Beispiel Initialisierung:

(*Init ST08_180_M1 Abstapeln*)
ST08_180_M1.sConfig.Description		:='Abstapeln';
ST08_180_M1.sConfig.InstName			:='ST08_180_M1';
ST08_180_M1.sConfig.Aktiv				:=TRUE;
ST08_180_M1.sConfig.Skalierfaktor		:=0.00034332275390625	;	(*360 / 1048576*)
ST08_180_M1.sConfig.Getriebefaktor		:=10;
ST08_180_M1.sConfig.Modulo			:=FALSE;
ST08_180_M1.sConfig.Pos_Faktor		:=5;				(*Weg bei einer Umdrehung in mm (nach Getriebe)*)
ST08_180_M1.sConfig.maxRpm			:=5338;
ST08_180_M1.sConfig.ModeOfOperation	:=CSP;			(*CSP,CSV,CST,CSTCA muss an der KLemme (Coe-Online 7010.03) eingestellt werden*)
(*nur für Coe-Online 7010.03 (CSP) position mode*)
ST08_180_M1.sConfig.RampTime		:=t#500ms;		(*Bauselle*)(*Beschleunigung und Bremsrampe*)
ST08_180_M1.sConfig.PosDiffControl_on	:=FALSE;		(*Baustelle*)
ST08_180_M1.sConfig.max_PosDiff		:=720;			(*Baustelle*)
ST08_180_M1.sConfig.SW_Limit_on		:=FALSE;
ST08_180_M1.sConfig.SW_Limit_min		:=-1000;
ST08_180_M1.sConfig.SW_Limit_max	:=1000;
ST08_180_M1.sConfig.lr_kp 				:= 800;
ST08_180_M1.sConfig.lr_ki 				:= 100.0;
ST08_180_M1.sConfig.lr_kd 				:= 50;

Beispiel Aufruf::

(*Call ST08_180_M1 Abstapeln*)
ST08_180_M1			(	sVisu:=	Visu.ST08_180_M1,
						Override:=	 MP.ST08.Override_Abstapeln,
						Offset:=		MP.ST08.PosOffsetAbstapeln.Pos,	(* in mm oder Grad am Abtrieb*)
						Reset:=		Visu.ModeSelect.BtnReset.Pressed );
IF	ST08_180_M1.sVisuAxis.BtnTeach.Pressed THEN
	TD.PosAbstapeln[ST08_180_M1.sVisuAxis.PosNr].Pos:= ST08_180_M1.sctrl.in.Position;
END_IF


 ===============================================================================================================================*)
END_ACTION
ACTION sub_connect:
IF	e_Toggle <> sHelp.b_ToggleHelp OR	(*die alten EL7211 haben kein e_Toggle, desshalb gibt es auch den e_State*)
	e_State = 8 THEN
	Connect:=TRUE;
	sHelp.b_ToggleHelp:=e_Toggle;
ELSE
	Connect:=FALSE;
END_IF
e_State:=e_State;(*
0x___1 = Slave in 'INIT' state
0x___2 = Slave in 'PREOP' state
0x___3 = Slave in 'BOOT' state
0x___4 = Slave in 'SAFEOP' state
0x___8 = Slave in 'OP' state
0x001_ = Slave signals error
0x002_ = Invalid vendorId, productCode... read
0x004_ = Initialization error occurred
0x008_ = Slave disabled
0x010_ = Slave not present
0x020_ = Slave signals link error
0x040_ = Slave signals missing link
0x080_ = Slave signals unexpected link
0x100_ = Communication port A
0x200_ = Communication port B
0x400_ = Communication port C
0x800_ = Communication port D*)
END_ACTION
ACTION sub_ctrl:
(*================================================================================================*)
(*Statusword*)
(*Bit  0*) sCtrl.in.Ready_to_switch_on:=		e_Statusword.0;
(*Bit 1 *) sCtrl.in.Switched_on:=			e_Statusword.1;
(*Bit 2 *) sCtrl.in.Operation_enabled	:=	e_Statusword.2;
(*Bit 3 *) sCtrl.in.Fault:=					e_Statusword.3;
(*Bit 4 *) 								e_Statusword.4;
(*Bit 5 *) 								e_Statusword.5;
(*Bit 6 *) sCtrl.in.Switch_on_disabled:=		e_Statusword.6;
(*Bit 7 *) sCtrl.in.Warning:=				e_Statusword.7;
(*Bit 8 *) 								e_Statusword.8;
(*Bit 9 *) 								e_Statusword.9;
(*Bit 10*) sCtrl.in.TxPDOToggle:=			e_Statusword.10; (*An-/Abwahl über 0x8010:01[} 136]*)
(*Bit 11*) sCtrl.in.Internal_Limit_active:=		e_Statusword.11;
(*Bit 12*) sCtrl.in.Target_value_ignored:=	e_Statusword.12;
(*Bit 13*) 								e_Statusword.13;
(*Bit 14*) 								e_Statusword.14;
(*Bit 15*) 								e_Statusword.15;

(*Controlword*)
(*Bit 0 *) a_Controlword.0:= sCtrl.out.Switch_on;
(*Bit 1 *) a_Controlword.1:= sCtrl.out.Enable_voltage;
(*Bit 2 *) a_Controlword.2:= sCtrl.out.Shutdown;
(*Bit 3 *) a_Controlword.3:= sCtrl.out.Enable_operation;
(*Bit 4 *) a_Controlword.4;
(*Bit 5 *) a_Controlword.5;
(*Bit 6 *) a_Controlword.6;
(*Bit 7 *) a_Controlword.7:= sCtrl.out.Fault_reset;
(*Bit 8 *) a_Controlword.8;
(*Bit 9 *) a_Controlword.9;
(*Bit 10*) a_Controlword.10;
(*Bit 11*) a_Controlword.11;
(*Bit 12*) a_Controlword.12;
(*Bit 13*) a_Controlword.13;
(*Bit 14*) a_Controlword.14;
(*Bit 15*) a_Controlword.15;
END_ACTION
ACTION sub_fb:
(* Zeiten *)
sFb.ton_uez		(IN:= ,PT:= t#3000ms, Q=>, ET=> );

sFb.ton_uez_velo	(IN:= sVelo.dif >15 AND on, PT:= t#300ms, Q=> , ET=> );
sFb.r_trig_Auto(CLK:=ModeSelect.Mode>MODE_MANUAL);
sFb.r_trig_Hand(CLK:=ModeSelect.Mode=MODE_MANUAL);
IF	sFb.r_trig_Hand.Q THEN
	sVisuAxis.Control:=TRUE;
ELSIF
	sFb.r_trig_Auto.Q THEN
	sVisuAxis.Control:=FALSE;
END_IF

(* Flanken *)
sFb.r_trig_stop(CLK:= NOT sVisuAxis.BtnStop.Pressed );
sFb.r_trig_reset(CLK:=NOT sVisuAxis.BtnReset.Pressed );
sFb.r_trig_MotorOn(CLK:=NOT sVisuAxis.BtnMotorOn.Pressed);
sFb.r_trig_jogP(CLK:= NOT sVisuAxis.BtnJogP.Pressed);
sFb.r_trig_jogM(CLK:=NOT sVisuAxis.BtnJogM.Pressed);
sFb.r_trig_MoveP(CLK:= NOT MoveP);
sFb.r_trig_MoveM(CLK:=NOT MoveN);
sFb.r_trig_MoveAbs(CLK:= NOT sVisuAxis.BtnMoveAbs.Pressed);

(*
sFb.ton_quitt		(IN:= ,PT:= t#100ms, Q=> , ET=> );
sFb.r_trig_quitt(CLK:=
			NOT On AND (*FEHLER wird dadurch automatisch quittiert*)
			NOT Reset AND
			NOT sVisuAxis.BtnReset.Pressed );
*)


sFb.ton_quitt(
		IN:=	NOT On AND (*FEHLER wird dadurch automatisch quittiert*)
				NOT Reset AND
				NOT sVisuAxis.BtnReset.Pressed ,
		PT:= 	t#200ms);
sFb.r_trig_quitt(CLK:=sFb.ton_quitt.Q);
END_ACTION
ACTION sub_Pos:
sPos.ist:=sctrl.in.Position;
(*===============================================================================*)
IF	(*config.Modulo OR*)
	sConfig.Pos_Faktor=0 THEN
	sConfig.Pos_Faktor:=1;
END_IF

(*Encoderüberlauf===================================================================================*)
sPos.lr_delta_ueberlauf:=ABS(sPos.lr_akt_alt - e_Position);

IF	sPos.lr_akt_alt >	(sPos.r_32bit - sPos.lr_delta_ueberlauf) AND						(*Überlauf bei 4294967295*)
	e_Position < sPos.lr_delta_ueberlauf THEN
	sPos.i32_count_ueberlauf:=	sPos.i32_count_ueberlauf +1;
ELSIF sPos.lr_akt_alt < sPos.lr_delta_ueberlauf AND									(*Überlauf bei 4294967295*)
	e_Position >(sPos.r_32bit - sPos.lr_delta_ueberlauf) THEN
	sPos.i32_count_ueberlauf:=	sPos.i32_count_ueberlauf -1;
END_IF
sPos.lr_akt_alt:= e_Position;

sPos.lr_Uebrlauf_Dist:=sPos.r_32bit * sConfig.Skalierfaktor;							(*Pos in Grad am Motor*)
sPos.lr_Uebrlauf_Dist:=sPos.lr_Uebrlauf_Dist/ sConfig.Getriebefaktor;					(*Pos in Grad am Getriebe*)

IF	NOT sConfig.Modulo THEN
	sPos.lr_Uebrlauf_Dist:=sPos.lr_Uebrlauf_Dist * (sConfig.Pos_Faktor/360);			(* Position in mm bei Linearachse*)
END_IF
sPos.lr_Uebrlauf_DistOne:=sPos.lr_Uebrlauf_Dist;

(*Positon auf Null stellen wenn der Überlauf erreicht ist*)
IF	sPos.i32_count_ueberlauf < - sConfig.Getriebefaktor THEN
	sCtrl.out.Target_Position:=sCtrl.out.Target_Position + (sConfig.Getriebefaktor * sPos.lr_Uebrlauf_DistOne );
	sPos.i32_count_ueberlauf:=sPos.i32_count_ueberlauf + LREAL_TO_DINT(sConfig.Getriebefaktor);
ELSIF  sPos.i32_count_ueberlauf >  sConfig.Getriebefaktor THEN
	sCtrl.out.Target_Position:=sCtrl.out.Target_Position - (sConfig.Getriebefaktor * sPos.lr_Uebrlauf_DistOne );
	sPos.i32_count_ueberlauf:=sPos.i32_count_ueberlauf - LREAL_TO_DINT(sConfig.Getriebefaktor);
END_IF

sPos.lr_Uebrlauf_Dist:=sPos.lr_Uebrlauf_Dist *DINT_TO_LREAL(sPos.i32_count_ueberlauf);

(*Multiturn======================================================================================*)

sConfig.Skalierfaktor;
sCtrl.in.Position:=UDINT_TO_LREAL(e_Position )*sConfig.Skalierfaktor;	(*Pos in Grad am Motor*)
(*sPos.lr_Mod:=LMOD(sCtrl.in.Position ,config.Modulofaktor);		(*Moduloposition*)*)
sCtrl.in.Position:=sCtrl.in.Position/ sConfig.Getriebefaktor;					(*Pos in Grad am Getriebe*)
sPos.lr_Mod:=LMOD((sCtrl.in.Position-Offset) ,360);			(*Pos in Grad 0° - 360° *)

IF	NOT sConfig.Modulo THEN
	sCtrl.in.Position:=sCtrl.in.Position * (sConfig.Pos_Faktor/360);			(* Position in mm bei Linearachse*)

	sPos.lr_Target:=sCtrl.out.Target_Position / (sConfig.Pos_Faktor/360) ;	(*Pos in Grad am Getriebe° *)
	sPos.lr_Offset_Ink:=Offset / (sConfig.Pos_Faktor/360) ;		 (*OffsetPos in Grad am Getriebe° *)
ELSE
	sPos.lr_Target:=sCtrl.out.Target_Position;
END_IF

sCtrl.in.Position:=sPos.lr_Uebrlauf_Dist+sCtrl.in.Position-Offset;

sPos.lr_Target:=sPos.lr_Target * sConfig.Getriebefaktor;				(*Pos in Grad am Motor° *)
sPos.lr_Offset_Ink:=sPos.lr_Offset_Ink* sConfig.Getriebefaktor;			(*OffsetPos in Grad am Motor° *)
sPos.i32_Offset_Ink:=LREAL_TO_UDINT(sPos.lr_Offset_Ink / sConfig.Skalierfaktor);		(*OffsetPos in Inkrementen am Motor° *)
a_Target_Position:=LREAL_TO_UDINT(sPos.lr_Target / sConfig.Skalierfaktor);	(*Pos in Inkrementen am Motor° *)

a_Target_Position:=a_Target_Position-sPos.i32_Offset_Ink;
e_Position;


(*Singelturn===Baustelle========================================================================*)
sPos.lr_ModuloPosInc:=LMOD(e_Position ,sPos.r_20bit);			(*Moduloposition in Ikrementen*)

sPos.lr_ModuloHelp:=(e_Position - LREAL_TO_UDINT(sPos.lr_ModuloPosInc)) / LREAL_TO_UDINT(sPos.r_20bit) ;
sPos.lr_ModuloHelp2:=(e_Position - LREAL_TO_UDINT(sPos.lr_ModuloPosInc)) / LREAL_TO_UDINT(sPos.r_20bit) ;
sPos.i16_ModuloHelp:=GANZE_ZAHL(sPos.lr_ModuloHelp2 / sConfig.Getriebefaktor);
sPos.lr_ModuloCount:=sPos.lr_ModuloHelp2 - (sPos.i16_ModuloHelp * sConfig.Getriebefaktor);

sPos.lr_Pos:= (sPos.lr_ModuloCount * sPos.r_20bit)+sPos.lr_ModuloPosInc;
sPos.lr_Pos:=sPos.lr_Pos* sConfig.Skalierfaktor;				(*Pos in Grad am Motor*)
sPos.lr_Pos:=sPos.lr_Pos / sConfig.Getriebefaktor;				(*Pos in Grad am Getriebe*)
sPos.lr_Pos:=LMOD(sPos.lr_Pos ,360);							(*Pos in Grad 0° - 360° *)
sPos.lr_Pos:=sPos.lr_Pos * (sConfig.Pos_Faktor/360);			(* Position in mm bei Linearachse*)



(*Schleppfehler===================================================================================*)
sCtrl.in.Following_Error:=DINT_TO_LREAL(e_Following_Error)*sConfig.Skalierfaktor;

sFb.ton_aufPos(
		IN:= ABS(sCtrl.out.Target_Position - sCtrl.in.Position) <1,
		PT:=t#20ms,
		Q=>On_Position);
END_ACTION
ACTION sub_rec_Torque:
IF	ABS(e_Torque) > Torque[1] THEN
	i:=1;
	FOR i:=NO_OF_Torque TO 2 BY-1 DO
	   Torque[i] := Torque[i-1];
	END_FOR
	 Torque[1]:=ABS(e_Torque);
END_IF
END_ACTION
ACTION sub_Regler:
sPos.r_18bit;
sVelo.Faktor:=sPos.r_18bit / 60;
(*=============================================================================================================*)

sVelo.maxRpmNachGertiebe	:=sConfig.maxRpm/ sConfig.Getriebefaktor;		(*Maximale Drehzahl nach Getriebe*)
sVelo.maxLinear		:=sVelo.maxRpmNachGertiebe * sConfig.Pos_Faktor;		(*Maximale Geschwindigkeit in mm/min*)
IF	 sConfig.Modulo THEN
	sVelo.maxRpm:=sVelo.maxRpmNachGertiebe;	(*rpm*)
	sVelo.Vorgabe_Velo_rpm:=Vorgabe_Velo * LREAL_TO_INT(sConfig.Getriebefaktor);
ELSE
	sVelo.maxRpm:=sVelo.maxLinear;			(*mm/min*)
	sVelo.Vorgabe_Velo_rpm:=Vorgabe_Velo / sConfig.Pos_Faktor;
	sVelo.Vorgabe_Velo_rpm:=sVelo.Vorgabe_Velo_rpm * LREAL_TO_INT(sConfig.Getriebefaktor);
END_IF

IF	Vorgabe_Velo > sVelo.maxRpm THEN
	Vorgabe_Velo:= LREAL_TO_INT(sVelo.maxRpm);
END_IF

sRegler.lr_Override:=DINT_TO_LREAL(override)/100;
sVelo.ist:=e_Velocity / sVelo.Faktor;				(*rpm am Motor*)
sVelo.ist:=sVelo.ist / sConfig.Getriebefaktor;		(*rpm nach Getriebe*)
sVelo.soll:=sVelo.sollRpm / sConfig.Getriebefaktor;	(*rpm nach Getriebe*)
IF	 NOT sConfig.Modulo THEN
	sVelo.ist:=sVelo.ist * sConfig.Pos_Faktor;		(*Geschwindigkeit in mm/min*)
	sVelo.soll:=sVelo.soll * sConfig.Pos_Faktor;	(*Geschwindigkeit in mm/min*)
END_IF

sVelo.dif:=									(*rpm oder mm*)
	ABS(sVelo.soll-sVelo.ist);

IF 	NOT sHelp.b_init2 AND sVelo.maxRpm<>0 THEN
	Vorgabe_Velo:=LREAL_TO_DINT(sVelo.maxRpm);
	sHelp.b_init2:=TRUE;
END_IF
sCtrl.in.Velocity:=sVelo.ist;
(*=============================================================================================================*)
CASE	sConfig.ModeOfOperation OF

CSV:
	sVelo.sollRpm:=LREAL_TO_INT(sVelo.Vorgabe_Velo_rpm * sRegler.lr_Override);

CSP:

	sRegler.lr_delta :=
			sCtrl.out.Target_Position -
			sCtrl.in.Position; (* Grad *)
	sRegler.lr_delta :=	sRegler.lr_delta * sConfig.Getriebefaktor;
	IF	NOT sConfig.Modulo THEN
 		sRegler.lr_delta:=sRegler.lr_delta / (sConfig.Pos_Faktor/360);
	END_IF

	sRegler.lr_tmp := sRegler.lr_delta;
	IF (sRegler.lr_tmp > 10000) THEN
		sRegler.lr_tmp := 10000;
	END_IF
	IF (sRegler.lr_tmp < -10000) THEN
		sRegler.lr_tmp := -10000;
	END_IF

	sRegler.lr_current_p := 0.004  * sConfig.lr_kp * sRegler.lr_tmp ; (*  RPM *)
	sRegler.lr_current_i := sRegler.lr_current_i + 0.004  * sConfig.lr_ki * sRegler.lr_tmp ; (*  RPM *)
	sRegler.lr_current_d := 0.004  * sConfig.lr_kd * (sRegler.lr_tmp-sRegler.lr_delta_alt) ; (*  RPM *)

	IF (sRegler.lr_current_i > 1000) THEN
		sRegler.lr_current_i := 1000;
	END_IF
	IF (sRegler.lr_current_i < -1000) THEN
		sRegler.lr_current_i := -1000;
	END_IF
	(*----------------------------------------------------------*)
	sRegler.lr_delta_dif:=sRegler.lr_delta_alt - sRegler.lr_delta;
	sPos.lr_DiffPuls:=ABS(sRegler.lr_delta_dif) ;
	sPos.lr_DiffPuls:=sPos.lr_DiffPuls*sConfig.Skalierfaktor;
	sPos.lr_DiffVelo:=ABS(sVelo.sollRpm/60*360/1000*4);
	(*sPos.lr_DiffPuls:=sPos.lr_DiffPuls-sPos.lr_DiffVelo;*)

	IF	sPos.lr_MaxDiff < sPos.lr_DiffPuls THEN
		sPos.lr_MaxDiff := sPos.lr_DiffPuls;
	END_IF
	IF	sPos.lr_DiffPuls = 0 AND on THEN
		sPos.lr_MaxDiff := 0;
	END_IF
	(*----------------------------------------------------------*)

	IF	sRegler.lr_targetpos_alt<>sCtrl.out.Target_Position THEN
		sRegler.lr_delta_targetpos:=ABS(sRegler.lr_targetpos_alt - sCtrl.out.Target_Position);
		sRegler.lr_targetpos_alt:=sCtrl.out.Target_Position;
		sFb.ton_aufPos.IN:=FALSE;
	END_IF

	(*----------------------------------------------------------*)

	sRegler.lr_delta_alt :=sRegler.lr_tmp;

	sRegler.lr_current_v :=sRegler.lr_current_p +sRegler.lr_current_i +sRegler.lr_current_d;
	sVelo.Vorgabe_Velo_rpm;
	IF (sRegler.lr_current_v >sVelo.Vorgabe_Velo_rpm) THEN
		sRegler.lr_current_v := sVelo.Vorgabe_Velo_rpm;
	ELSIF (sRegler.lr_current_v < -sVelo.Vorgabe_Velo_rpm) THEN
		sRegler.lr_current_v := -sVelo.Vorgabe_Velo_rpm;
	END_IF

	sRegler.lr_current_v :=sRegler.lr_current_v ;

	IF	sRegler.lr_delta_targetpos >= 360 THEN
		IF	(ABS(sRegler.lr_delta) < 360) THEN
			sRegler.lr_current_v :=sRegler.lr_current_v * (ABS(sRegler.lr_delta) / 360);
		END_IF
	ELSE
		sRegler.lr_current_v := sRegler.lr_current_v * (ABS(sRegler.lr_delta) / 180);
	END_IF
	IF 	On_Position THEN
		sRegler.lr_delta_targetpos := 360;
	END_IF

	sVelo.sollRpm := LREAL_TO_DINT(sRegler.lr_current_v);

END_CASE


(*Beschränken auf Vorgabe*)

IF	sVelo.sollRpm > sVelo.Vorgabe_Velo_rpm THEN
	sVelo.sollRpm :=LREAL_TO_INT(sVelo.Vorgabe_Velo_rpm);
END_IF

IF	sVelo.sollRpm < sVelo.Vorgabe_Velo_rpm*(-1) THEN
	sVelo.sollRpm :=LREAL_TO_INT(sVelo.Vorgabe_Velo_rpm*(-1));
END_IF

sVelo.sollRpm:=sVelo.sollRpm * sRegler.lr_Override;

(*Ausgaber an Regler*)
IF 	on THEN
	a_Target_Velocity:=
		LREAL_TO_DINT(
		sVelo.sollRpm *
		 sVelo.Faktor) ;
ELSE
	a_Target_Velocity:=0;
END_IF
e_Velocity;
END_ACTION
ACTION sub_sdo:
(*=============================================================================================*)
sSdo.s_SlaveNetId:='172.18.137.69.4.1';
sSdo.ui16_SlaveAddr:=1012;
sSdo.i8_SubIndex:=0;
sSdo.w_Index:=16#8000;

(* Einen neuen EcCoeSdo-Parameter auf den Antrieb schreiben *)
sSdo.fb_ec_coe_sdo_write_ex(
	sNetId:= sSdo.s_SlaveNetId,
	nSlaveAddr:= sSdo.ui16_SlaveAddr,
	nSubIndex:= sSdo.i8_SubIndex,
	nIndex:= sSdo.w_Index,
	pSrcBuf:= ADR(sSdo.acObjectData),
	cbBufLen:= SIZEOF(sSdo.acObjectData),
	bExecute:= ,
	tTimeout:= t#10s,
	bCompleteAccess:= FALSE,
	bBusy=> ,
	bError=> ,
	nErrId=> );

(*=============================================================================================*)
(* Einen neuen EcCoeSdo-Parameter von dem Antrieb lesen *)
sSdo.fb_ec_coe_sdo_read_ex(
	sNetId:= sSdo.s_SlaveNetId,
	nSlaveAddr:= sSdo.ui16_SlaveAddr,
	nSubIndex:= sSdo.i8_SubIndex,
	nIndex:= sSdo.w_Index,
	pDstBuf:=  ADR(sSdo.acObjectData),
	cbBufLen:= SIZEOF(sSdo.acObjectData),
	bExecute:= ,
	tTimeout:= t#10s,
	bCompleteAccess:= FALSE,
	bBusy=> ,
	bError=> ,
	nErrId=> );
END_ACTION
ACTION sub_Visu:
sFb.r_trig_kont(CLK:= sVisuAxis.b_kont, Q=> );
sFb.r_trig_ink_10(CLK:= sVisuAxis.b_ink_10, Q=> );
sFb.r_trig_ink_100(CLK:= sVisuAxis.b_ink_100, Q=> );
sFb.r_trig_ink_1000(CLK:= sVisuAxis.b_ink_1000, Q=> );
sFb.r_trig_ink_var(CLK:= sVisuAxis.b_ink_var, Q=> );

IF	sFb.r_trig_kont.Q THEN
	sVisuAxis.b_ink_10:=FALSE;
	sVisuAxis.b_ink_100:=FALSE;
	sVisuAxis.b_ink_1000:=FALSE;
	sVisuAxis.b_ink_var:=FALSE;
ELSIF
	sFb.r_trig_ink_10.Q THEN
	sVisuAxis.b_kont:=FALSE;
	sVisuAxis.b_ink_100:=FALSE;
	sVisuAxis.b_ink_1000:=FALSE;
	sVisuAxis.b_ink_var:=FALSE;
ELSIF
	sFb.r_trig_ink_100.Q THEN
	sVisuAxis.b_kont:=FALSE;
	sVisuAxis.b_ink_10:=FALSE;
	sVisuAxis.b_ink_1000:=FALSE;
	sVisuAxis.b_ink_var:=FALSE;
ELSIF
	sFb.r_trig_ink_1000.Q THEN
	sVisuAxis.b_kont:=FALSE;
	sVisuAxis.b_ink_10:=FALSE;
	sVisuAxis.b_ink_100:=FALSE;
	sVisuAxis.b_ink_var:=FALSE;
ELSIF
	sFb.r_trig_ink_var.Q THEN
	sVisuAxis.b_kont:=FALSE;
	sVisuAxis.b_ink_10:=FALSE;
	sVisuAxis.b_ink_100:=FALSE;
	sVisuAxis.b_ink_1000:=FALSE;
ELSIF
	NOT sVisuAxis.b_kont AND
	NOT sVisuAxis.b_ink_10  AND
	NOT sVisuAxis.b_ink_100 AND
	NOT sVisuAxis.b_ink_1000 AND
	NOT sVisuAxis.b_ink_var THEN
	sVisuAxis.b_kont:=TRUE;
END_IF


IF	(sFb.r_trig_jogP.Q OR sFb.r_trig_jogM.Q) AND
	NOT sVisuAxis.b_kont THEN

	IF	sVisuAxis.b_ink_10  THEN
		Vorgabe_Pos_Rel:=0.01;
	ELSIF
		sVisuAxis.b_ink_100 THEN
		Vorgabe_Pos_Rel:=0.1;
	ELSIF
		sVisuAxis.b_ink_1000 THEN
		Vorgabe_Pos_Rel:=1;
	ELSIF
		sVisuAxis.b_ink_var THEN
		Vorgabe_Pos_Rel:=sVisuAxis.lr_ink_var;
	END_IF

	IF	sFb.r_trig_jogM.Q THEN
		Vorgabe_Pos_Rel:=Vorgabe_Pos_Rel * (-1);
	END_IF
	MoveRel:=TRUE;
END_IF

(*Positon aktivieren=======================================================*)
FOR i := -1 TO NO_OF_POS_AXIS  BY 1DO
	IF	sVisuAxis.b_Pos_nr[i] THEN
		sVisuAxis.PosNr:=i;
		Vorgabe_Pos_Abs:=sPosList[i].Pos;
	END_IF
END_FOR
sVisuAxis.b_Pos_nr:=sHelp.b_Pos_nr_Empty;


IF	sHelp.Pos <> sPosList[sVisuAxis.PosNr].Pos OR
	sHelp.PosNr <> sVisuAxis.PosNr OR
	 sVisuAxis.b_PosNr THEN
	Vorgabe_Pos_Abs:=sPosList[sVisuAxis.PosNr].Pos;
END_IF
sHelp.PosNr:=sVisuAxis.PosNr;
sHelp.Pos:=sPosList[sVisuAxis.PosNr].Pos;
END_ACTION

(* POU zLibrary/ept/Achse/GANZE_ZAHL, ST *)
FUNCTION GANZE_ZAHL : INT
VAR_INPUT
	lr_Wert		:LREAL;
END_VAR
VAR
	st_Wert		:STRING;
	pos			:INT;
END_VAR
IF	lr_Wert >= 1 THEN

	st_Wert:=LREAL_TO_STRING(lr_Wert);
	pos:=FIND(st_Wert,'.');
	
	st_Wert:=LEFT(st_Wert,pos);
	
	GANZE_ZAHL:=STRING_TO_INT(st_Wert);
ELSE
	GANZE_ZAHL:=0;
END_IF
END_FUNCTION

(* POU zLibrary/ept/Achse/fb_Auto_On_Off, ST *)
FUNCTION_BLOCK fb_Auto_On_Off
VAR_INPUT
	b_Stop				:BOOL;
END_VAR
VAR_IN_OUT
	Achse				:fb_72x1_Achse;
END_VAR
VAR
	fb_ton_wz			:TON;
	fb_ton_uez			:TON;

	fb_state_entry		:ST_StateEntry;
END_VAR
fb_ton_wz		(IN:= ,PT:= , Q=>  , ET=> );
fb_ton_uez		(IN:= ,PT:= t#2000ms, Q=>, ET=> );

(* ==================================Schrittkette================================ *)
fb_state_entry(	i16_pos:= 1);

CASE fb_state_entry.i16_step OF
(*=======================================================*)
INIT_OBJ:
	fb_state_entry.i16_next_step := INIT;

(*==========================================================================================================*)
INIT:
	fb_state_entry.i16_next_step := BEREIT;

(*==========================================================================================================*)
BEREIT:
	IF	fb_state_entry.E THEN
		;
	END_IF

	IF	ModeSelect.Mode=MODE_AUTO OR
		ModeSelect.Mode=MODE_AUTO_RUN OR
		ModeSelect.Mode=MODE_STEP_RUN THEN

		IF	NOT Achse.On AND
			NOT b_Stop AND
			NOT Achse.Error_ THEN
			Achse.MotorOn:=TRUE;
		END_IF

		fb_ton_uez.IN:=Achse.MotorOn;

		IF	b_Stop AND Achse.MotorOn THEN
			Achse.MotorOn:=FALSE;
			Achse.MotorOff:= TRUE;
		END_IF

	END_IF

(*==========================================================================================================*)
FEHLER: (*Fehler*)
	IF	fb_state_entry.E THEN
		;
	END_IF

END_CASE

fb_state_entry(i16_pos:= 2);
END_FUNCTION_BLOCK

(* POU zLibrary/ept/BDE/Fb_ExportHydraString, ST *)
FUNCTION_BLOCK Fb_ExportHydraString
VAR_INPUT
	s_Path				: T_MaxString;
	s_system_time		: STRING;
	st_data				: struct_Hydra8;
	bKopiereDateiAufServer	: BOOL := FALSE;
	sDateiName			: STRING := 'Eingang.txt';
	tStartTime			: TIME := T#10S;
	sToolPath			: STRING(255) := '';
END_VAR
VAR
	fb_state_entry			: ST_StateEntry;
	fbFindFiles			: FB_EnumFindFileList;
	fbFindFilesEntry		: ST_FindFileEntry;
	fbFileOpen			: FB_FileOpen;
	fbFilePuts			: FB_FilePuts;
	fbFileClose			: FB_FileClose;
	HelpString			: T_MaxString;
	Substring			:ARRAY[1..3] OF STRING(255);
	fb_ton_start			: TON;
	hFile					:UINT;
	nErrIdOpen					:UDINT;
	nErrIdWrite					:UDINT;
	nErrIdClose					:UDINT;
	nErrIdCloseCounter			:UDINT;
	sFileName				:STRING;
	i						:UINT;

	i_dint_to_hydra		: DINT;
	s_dint_to_hydra	: STRING;

	sDatum		: STRING(10) := '01/01/1970';	(* aktuelles Datum im Format TT/MM/JJJJ *)
	sZeit		: STRING(8) := '00:00:00';	(* aktuelle Zeit im Format HH:MM:SS *)

	sPathStrDateiAufServerSpeichern	:T_MaxString;	(* Pfad damit Leerzeichen im Pfad erlaubt sind*)
	DateiAufServerSpeichern 		:NT_StartProcess;
END_VAR
VAR_OUTPUT
	Ready						:BOOL;
	Busy						:BOOL;
	Done						:BOOL;
	Error						:BOOL;
END_VAR
VAR CONSTANT
	sMSTAT					: STRING := 'MSTAT=';
	sDatumPrefix				: STRING := 'DAT=';
	sZeitPrefix				: STRING := 'ZEI=';
	sCounter					: STRING := 'COUNTER';
	sTrennzeichen			: STRING := '|';
	sDosGeraetePfad			: STRING(4) := '\\.\';	(* https://docs.microsoft.com/de-de/dotnet/standard/io/file-path-formats
	Das Windows-Betriebssystem verfügt über ein einheitliches Objektmodell,
	das auf alle Ressourcen, einschließlich Dateien, verweist. Sie können über
	das Konsolenfenster auf diese Objektpfade zugreifen. Diese werden über einen
	speziellen Ordner aus symbolischen Verknüpfungen, denen ältere DOS- und UNC-Pfade
	zugeordnet sind, für die Win32-Schicht zur Verfügung gestellt. Der Zugriff auf
	diesen speziellen Ordner erfolgt über die DOS-Gerätepfadsyntax, die einer der Folgenden entspricht:*)
END_VAR
(*======================================================
   FB: Fb_ExportHydraString
 ------------------------------------------------------
   Auth: 	Thomas Vilgis    						 
   Date: 	27.01.2022    						     
   Rev.: 		1.1	
   Desc:		Dieser Baustein übernimmt die Kommunikation zum neuen Hydra 8.
			Es wird alle 2 Sekunden (Zeit einstellbar) eine Textdatei mit den Produktionsdaten für
			das Hydra erstellt. Hydra liest diese Datei aus und löscht sie dann.
			Alle Daten werden in eine Zeile geschrieben
			Es gibt insgesamt 20 Zähler. Es werden aber nur die jeweils 4 letzten Ziffern übergeben.
			Fehlende Ziffern werden mit 0 aufgefüllt.
			Dann gibt es noch 999 Status-Bits. Das erste TRUE-Bit im  Array wird als Status übergeben.
			Außerdem werden noch die aktuelle Uhrzeit und das Datum übergeben.
			Auf Wunsch von Stanzerei Augsburg wurde aus diesem Baustein ein Fb gemacht.
			Per Vbs-Stript wird eine Batch-Datei gestartet, die die erzeugte txt-Datei auf den
			Server verschiebt. Dort soll eine zusätzliche Auswertung durchgeführt werden.
			NEU: Neuaufbau FB, da Filehandle zu Fehlern führt (D.Peichl 16.02.2022)
   Historie: 	1.1

 ========================================================*)



(* Zeiten *)
fb_ton_start(IN:= NOT fb_ton_start.Q, PT:= tStartTime, Q=>  , ET=> );


(* ======================================Schrittkette======================================== *)
fb_state_entry(i16_pos:= 1);

CASE fb_state_entry.i16_step OF
(*=======================================================*)
	INIT_OBJ: fb_state_entry.s_debugtext:='initialisieren';	

		(*-----------------------Weiterschaltbedingungen----------------------------*)
		IF fb_state_entry.fb_ton_Step.ET >= T#5S THEN
			fb_state_entry.i16_next_step:=BEREIT;
		END_IF

		IF fb_state_entry.X THEN
			sFileName:=CONCAT(s_Path,sDateiName);
			sPathStrDateiAufServerSpeichern := CONCAT(sDosGeraetePfad, sToolPath);
		END_IF

(*=======================================================*)
	BEREIT: fb_state_entry.s_debugtext:='Start';

		IF fb_state_entry.E THEN
			Ready := TRUE;
		END_IF

		(*-----------------------Weiterschaltbedingungen----------------------------*)
		IF fb_ton_start.Q THEN
			Error := FALSE;
			Busy := TRUE;
			Ready := FALSE;
			Done := FALSE;
			fb_state_entry.i16_next_step:=110;
		END_IF

(*=======================================================*)
	110: fb_state_entry.s_debugtext:='Prüfe, ob Datei geschlossen ist';

		(*-----------------------Weiterschaltbedingungen----------------------------*)
		IF hFile = 0 THEN
			fb_state_entry.i16_next_step:=120;
		ELSE
			fb_state_entry.i16_next_step:=112;
		END_IF
		
(*=======================================================*)
	112: fb_state_entry.s_debugtext:='Datei schließen';

		IF fb_state_entry.E THEN
			fbFileClose.bExecute:=TRUE;
		END_IF

		(*-----------------------Weiterschaltbedingungen----------------------------*)
		IF 	fbFileClose.bBusy THEN
			fb_state_entry.i16_next_step:=114;
		END_IF

(*=======================================================*)
	114: fb_state_entry.s_debugtext:='Datei schließen';

		(*-----------------------Weiterschaltbedingungen----------------------------*)
		IF NOT fbFileClose.bBusy THEN
			hFile := 0;
			fbFileClose.bExecute:=FALSE;
			IF 	fbFileClose.bError THEN
				nErrIdClose:=fbFileClose.nErrId;
				nErrIdCloseCounter := nErrIdCloseCounter + 1;
				fb_state_entry.i16_next_step:=FEHLER;
			ELSE
				fb_state_entry.i16_next_step:=120;
			END_IF
		END_IF

(*=======================================================*)
	120: fb_state_entry.s_debugtext:='Prüfe, ob Datei vorhanden ist';

		IF fb_state_entry.E THEN
			fbFindFiles.bExecute := TRUE;
		END_IF

		(*-----------------------Weiterschaltbedingungen----------------------------*)
		IF fbFindFiles.bBusy THEN
			fb_state_entry.i16_next_step:=130;
		END_IF

(*=======================================================*)
	130: fb_state_entry.s_debugtext:='Prüfe, ob Datei vorhanden ist';

		(*-----------------------Weiterschaltbedingungen----------------------------*)
		IF NOT fbFindFiles.bBusy THEN
			fbFindFiles.bExecute := FALSE;
			IF NOT fbFindFiles.bError THEN
				IF fbFindFiles.nFindFiles = 0 THEN
					fb_state_entry.i16_next_step:=140;
				ELSE
					fb_state_entry.i16_next_step:=300;	(* Datei noch vorhanden >> tue nichts *)
				END_IF
			ELSE
				fb_state_entry.i16_next_step:=FEHLER;
			END_IF
		END_IF
		
(*=======================================================*)
	140: fb_state_entry.s_debugtext:='Counter 1-10 umwandeln und sezte Strings zusammen';

		IF fb_state_entry.E THEN
			Substring[1] := '';
			FOR i := 1 TO 10 BY 1 DO
				i_dint_to_hydra := st_data.iCounter[i];
				subr_Dint_to_Hydra_Counter();							(* Zähler in String umwandeln *)
				HelpString := CONCAT(sCounter, UINT_TO_STRING(i));
				HelpString := CONCAT(HelpString, '=');
				HelpString := CONCAT(HelpString, s_dint_to_hydra);
				HelpString := CONCAT(HelpString, sTrennzeichen);
				Substring[1] := CONCAT(Substring[1], HelpString);
			END_FOR
		END_IF

		(*-----------------------Weiterschaltbedingungen----------------------------*)
			fb_state_entry.i16_next_step:=142;
			
(*=======================================================*)
	142: fb_state_entry.s_debugtext:='Counter 10-20 umwandeln und sezte Strings zusammen';

		IF fb_state_entry.E THEN
			Substring[2] := '';
			FOR i := 11 TO 20 BY 1 DO
				i_dint_to_hydra := st_data.iCounter[i];
				subr_Dint_to_Hydra_Counter();							(* Zähler in String umwandeln *)
				HelpString := CONCAT(sCounter, UINT_TO_STRING(i));
				HelpString := CONCAT(HelpString, '=');
				HelpString := CONCAT(HelpString, s_dint_to_hydra);
				HelpString := CONCAT(HelpString, sTrennzeichen);
				Substring[2]:= CONCAT(Substring[2], HelpString);
			END_FOR
		END_IF

		(*-----------------------Weiterschaltbedingungen----------------------------*)
			fb_state_entry.i16_next_step:=144;
		
(*=======================================================*)
	144: fb_state_entry.s_debugtext:='Lese Daten und sezte Strings zusammen';

		IF fb_state_entry.E THEN
			(* Datum in das richtige Format bringen *)
			HelpString := MID(s_system_time, 2, 4);
			HelpString := CONCAT(HelpString, '/');
			HelpString := CONCAT(HelpString, MID(s_system_time, 2, 1));
			HelpString := CONCAT(HelpString, '/');
			HelpString := CONCAT(HelpString, MID(s_system_time, 4, 7));
			sDatum := HelpString;

			(* Zeit in das richtige Format bringen *)
			sZeit := MID(s_system_time, 8, 12);

			(* Prüfe welcher Status aktiv ist. Der niedrigste Status wird in Datei eingetragen *)
			FOR i := 1 TO 999 BY 1 DO
				IF st_data.bStatus[i] THEN
					EXIT;	(* Verlasse Schleife *)
				END_IF
			END_FOR

			(* wenn kein Status aktiv ist, dann schreibe MSTAT@M100=    Ohne Zahl  *)
			(* Falls kein Produktionssignal, dann Nicht zugeordnet *)
			IF i < 999 THEN
				HelpString := CONCAT(sMSTAT, UINT_TO_STRING(i));
			ELSE
				HelpString := 'MSTAT=30000';
			END_IF

			Substring[3] := '';
			HelpString := CONCAT(HelpString, sTrennzeichen);
			HelpString := CONCAT(HelpString, sDatumPrefix);
			HelpString := CONCAT(HelpString, sDatum);
			HelpString := CONCAT(HelpString, sTrennzeichen);
			HelpString := CONCAT(HelpString, sZeitPrefix);
			HelpString := CONCAT(HelpString, sZeit);
			Substring[3] := HelpString;
		END_IF

		(*-----------------------Weiterschaltbedingungen----------------------------*)
		fb_state_entry.i16_next_step:=150;
		
(*=======================================================*)
	150: fb_state_entry.s_debugtext:='Datei erstellen';

		IF fb_state_entry.E THEN
		   	fbFileOpen.bExecute:=TRUE;
		END_IF

		(*-----------------------Weiterschaltbedingungen----------------------------*)
		IF fbFileOpen.bBusy THEN
			fb_state_entry.i16_next_step:=160;
		END_IF

(*=======================================================*)
	160: fb_state_entry.s_debugtext:='Datei erstellen';

		(*-----------------------Weiterschaltbedingungen----------------------------*)
		IF 	NOT fbFileOpen.bBusy THEN
			i:=1;						(*wichtig für Dateizusammenbau*)
			fbFileOpen.bExecute:=FALSE;
			IF 	fbFileOpen.bError THEN
				nErrIdOpen:=fbFileOpen.nErrId;
				fb_state_entry.i16_next_step:=200;
			ELSE
				hFile := fbFileOpen.hFile;	(* Sehr wichtig hFile für FilePuts und Fileclose übergeben *)
				fb_state_entry.i16_next_step:=170;
			END_IF
		END_IF

(*=======================================================*)
	170: fb_state_entry.s_debugtext:='String in Datei eintragen';

		IF fb_state_entry.E THEN
			fbFilePuts.sLine:=Substring[i];
			fbFilePuts.bExecute:=TRUE;
		END_IF

		(*-----------------------Weiterschaltbedingungen----------------------------*)
		IF  fbFilePuts.bBusy THEN
			fb_state_entry.i16_next_step:=180;
		END_IF

(*=======================================================*)
	180: fb_state_entry.s_debugtext:='String in Datei eintragen';

		(*-----------------------Weiterschaltbedingungen----------------------------*)
		IF 	NOT fbFilePuts.bBusy THEN
			fbFilePuts.bExecute:=FALSE;
			IF 	fbFilePuts.bError THEN
				nErrIdWrite:=fbFilePuts.nErrId;
				fb_state_entry.i16_next_step:=200;
			ELSE
				fb_state_entry.i16_next_step:=190;
			END_IF
		END_IF

(*=======================================================*)
	190: fb_state_entry.s_debugtext:='Schleife Substrings in Datei eintragen';

		IF fb_state_entry.E THEN
			i :=  i+1;
		END_IF

		(*-----------------------Weiterschaltbedingungen----------------------------*)
		IF i <= 3 THEN
			fb_state_entry.i16_next_step:=170;
		ELSE
			fb_state_entry.i16_next_step:=200;
		END_IF

(*=======================================================*)
	200: fb_state_entry.s_debugtext:='Datei schließen';

		IF fb_state_entry.E THEN
			fbFileClose.bExecute:=TRUE;
		END_IF

		(*-----------------------Weiterschaltbedingungen----------------------------*)
		IF 	fbFileClose.bBusy THEN
			fb_state_entry.i16_next_step:=210;
		END_IF

(*=======================================================*)
	210: fb_state_entry.s_debugtext:='Datei schließen';

		(*-----------------------Weiterschaltbedingungen----------------------------*)
		IF NOT fbFileClose.bBusy THEN
			hFile := 0;
			fbFileClose.bExecute:=FALSE;
			IF 	fbFileClose.bError THEN
				nErrIdClose:=fbFileClose.nErrId;
				nErrIdCloseCounter := nErrIdCloseCounter + 1;
				fb_state_entry.i16_next_step:=FEHLER;
			ELSE
				fb_state_entry.i16_next_step:=300;
			END_IF
		END_IF

(*=======================================================*)
	300: fb_state_entry.s_debugtext:='Abfrage, kopiere Datei auf Server?';

		(*-----------------------Weiterschaltbedingungen----------------------------*)
		IF bKopiereDateiAufServer THEN
			fb_state_entry.i16_next_step:=310;
		ELSE
			Busy := FALSE;
			Done := TRUE;
			fb_state_entry.i16_next_step:=BEREIT;
		END_IF

(*=======================================================*)
	310: fb_state_entry.s_debugtext:='Kopiere Datei auf Server';

		IF fb_state_entry.E THEN
			DateiAufServerSpeichern.START := TRUE;
		END_IF

		(*-----------------------Weiterschaltbedingungen----------------------------*)
		IF DateiAufServerSpeichern.BUSY THEN
			fb_state_entry.i16_next_step:=320;
		ELSIF fb_state_entry.fb_ton_Step.ET >= T#2s THEN
			fb_state_entry.i16_next_step:=FEHLER;
		END_IF

		IF fb_state_entry.X THEN
			DateiAufServerSpeichern.START := FALSE;
		END_IF

(*=======================================================*)
	320: fb_state_entry.s_debugtext:='Warte bis fertig';

		(*-----------------------Weiterschaltbedingungen----------------------------*)
		IF NOT DateiAufServerSpeichern.BUSY AND
			NOT DateiAufServerSpeichern.ERR THEN
			fb_state_entry.i16_next_step:=330;
		ELSIF fb_state_entry.fb_ton_Step.ET >= T#5s THEN
			fb_state_entry.i16_next_step:=FEHLER;
		END_IF

(*=======================================================*)
	330: fb_state_entry.s_debugtext:='fertig';

		(*-----------------------Weiterschaltbedingungen----------------------------*)
		Busy := FALSE;
		Done := TRUE;
		fb_state_entry.i16_next_step:=BEREIT;

(*=======================================================*)
	FEHLER:
		IF fb_state_entry.E THEN
			Error := TRUE;
		END_IF

		(*-----------------------Weiterschaltbedingungen----------------------------*)
		fb_state_entry.i16_next_step:=BEREIT;

END_CASE


fb_state_entry(i16_pos:= 2);



fbFindFiles(
	bExecute	:= ,
	sNetId		:= '',
	sPathName	:= sFileName,
	pFindList	:= ADR(fbFindFilesEntry),
	cbFindList	:= SIZEOF(fbFindFilesEntry),
	tTimeout	:= t#15s );

 fbFileOpen(
	sNetId:='',
	sPathName:= sFileName,
	nMode:=FOPEN_MODEAPPEND,
	ePath:=PATH_GENERIC,
	bExecute:= ,
	tTimeout:=T#15s,
	hFile=> );

fbFilePuts(
	sNetId:='',
	hFile:=hFile,
	sLine:= ,
	bExecute:= ,
	tTimeout:=t#15s);

fbFileClose(
	sNetId:='',
	hFile:=hFile,
	bExecute:= ,
	tTimeout:=t#15s);

DateiAufServerSpeichern(
	NETID:='',
	PATHSTR	:='C:\Windows\System32\wscript.exe',
	DIRNAME	:=sPathStrDateiAufServerSpeichern,
	COMNDLINE	:='HydraDateiAufServerSpeichern.vbs',
	START		:=,
	TMOUT		:=T#10s);
END_FUNCTION_BLOCK
ACTION subr_Dint_to_Hydra_Counter:
(* Damit nur noch 4 Stellen übrig bleiben *)
i_dint_to_hydra := i_dint_to_hydra MOD 10000;

s_dint_to_hydra := DINT_TO_STRING(i_dint_to_hydra);
(* vordere Stellen mit 0 auffüllen *)
WHILE(LEN(s_dint_to_hydra) < 4) DO
	s_dint_to_hydra := CONCAT('0', s_dint_to_hydra);
END_WHILE
END_ACTION

(* POU zLibrary/ept/Checks/CheckBounds, ST *)
FUNCTION CheckBounds : DINT
VAR_INPUT
	index, lower, upper 	: DINT;
END_VAR
VAR
END_VAR
IF index<lower THEN
	CheckBounds_ErrCnt := CheckBounds_ErrCnt + 1;
	CheckBounds := lower;
ELSIF index>upper THEN
	CheckBounds_ErrCnt := CheckBounds_ErrCnt + 1;
	CheckBounds := upper;
ELSE
	CheckBounds := index;
END_IF
END_FUNCTION

(* POU zLibrary/ept/Checks/CheckDivByte, ST *)
FUNCTION CheckDivByte : BYTE
VAR_INPUT
	divisor			 	: BYTE;
END_VAR
VAR
END_VAR
IF divisor = 0 THEN
	CheckByteZeroDiv_ErrCnt := CheckByteZeroDiv_ErrCnt + 1;
	CheckDivByte := 1;
ELSE
	CheckDivByte := divisor;
END_IF
END_FUNCTION

(* POU zLibrary/ept/Checks/CheckDivDWord, ST *)
FUNCTION CheckDivDWord : DWORD
VAR_INPUT
	divisor				: DWORD;
END_VAR
VAR
END_VAR
IF divisor = 0 THEN
	CheckDWordZeroDiv_ErrCnt := CheckDWordZeroDiv_ErrCnt + 1;
	CheckDivDWord := 1;
ELSE
	CheckDivDWord := divisor;
END_IF
END_FUNCTION

(* POU zLibrary/ept/Checks/CheckDivReal, ST *)
FUNCTION CheckDivReal : REAL
VAR_INPUT
	divisor		 		: REAL;
END_VAR
VAR
END_VAR
IF divisor = 0 THEN
	CheckRealZeroDiv_ErrCnt := CheckRealZeroDiv_ErrCnt + 1;
	CheckDivReal := 1;
ELSE
	CheckDivReal := divisor;
END_IF
END_FUNCTION

(* POU zLibrary/ept/Checks/CheckDivWord, ST *)
FUNCTION CheckDivWord : WORD
VAR_INPUT
	divisor				: WORD;
END_VAR
VAR
END_VAR
IF divisor = 0 THEN
	CheckWordZeroDiv_ErrCnt:= CheckWordZeroDiv_ErrCnt + 1;
	CheckDivWord := 1;
ELSE
	CheckDivWord := divisor;
END_IF
END_FUNCTION

(* POU zLibrary/ept/Checks/CheckRangeSigned, ST *)
FUNCTION CheckRangeSigned : DINT
VAR_INPUT
    value, lower, upper: DINT;
END_VAR
VAR
END_VAR
IF (value < lower) THEN
	CheckRangeSigned_ErrCnt := CheckRangeSigned_ErrCnt + 1;
	CheckRangeSigned := lower;
ELSIF(value > upper) THEN
	CheckRangeSigned_ErrCnt := CheckRangeSigned_ErrCnt + 1;
	CheckRangeSigned := upper;
ELSE
	CheckRangeSigned := value;
END_IF
END_FUNCTION

(* POU zLibrary/ept/Checks/CheckRangeUnsigned, ST *)
FUNCTION CheckRangeUnsigned : UDINT
VAR_INPUT
    value, lower, upper: UDINT;
END_VAR
VAR
END_VAR
IF (value < lower) THEN
	CheckRangeUnSigned_ErrCnt := CheckRangeUnsigned_ErrCnt + 1;
	CheckRangeUnsigned := lower;
ELSIF(value > upper) THEN
	CheckRangeUnsigned_ErrCnt := CheckRangeUnsigned_ErrCnt + 1;
	CheckRangeUnsigned := upper;
ELSE
	CheckRangeUnsigned := value;
END_IF
END_FUNCTION

(* POU zLibrary/Keyence/FB_KeyenceEtherCat, ST *)
FUNCTION_BLOCK FB_KeyenceEtherCat
VAR_INPUT
	st_ctrl_in						: struct_ctrl_in;
	JobNo							: INT;
	sConfig							: st_config_Keyence;	(*Initialisierung der Kamera*)
END_VAR
VAR_OUTPUT
	st_ctrl_out						: struct_ctrl_out;
	Connected						: BOOL;
	ActJobNo						: INT;
	b_Kam_Pruef_IO				: BOOL; 				(* Kameraprüfung Ergebnis iO *)
	b_Kam_Pruef_NIO				: BOOL; 				(* Kameraprüfung Ergebnis niO *)
	RecvDataString					: T_MaxString;
END_VAR
VAR
	b_Test							: BOOL;

	fb_ton_quitt						: TON;
	fb_state_entry					: ST_StateEntry;

 	BtnConnect						: sButtonVisu;
	BtnTrigger						: sButtonVisu;

	sm_kamera_keine_reaktion		: BOOL := FALSE;
	sm_kamera_nicht_bb			: BOOL := FALSE;
	sm_jobnummer_nicht_erlaubt		: BOOL := FALSE;		(* erlaubter Bereich von 0-15 *)
	sm_kamera_controler_error		: BOOL := FALSE;

	i								: INT;
	nInByte							: BYTE;

	stControl						: st_ctrl_out_Keyence;

	FB_ReadXmlLineConf			: FB_ReadXmlLine;
	FB_ReadXmlLineMsg			: FB_ReadXmlLine;
	(*Variablen für Behr Meldungen*)
	TempErrorText					: STRING(255);
	ProcessTime					: DINT;				(* Counts the time in steps of 100ms since starting operation *)
	Error							: ErrorStruct;

(*DL-EC1A: PDO-Kommunikation (Prozessdaten-Objekte)*)

	(*Input Request*)
	anInputRequest					AT%Q* 	: ARRAY [0..4] OF DWORD;

	(*Status of System*)
	bError_Status_00				AT%I*	: BOOL;		(* *)
(*	nError_Code_00					AT%I*	: UINT;							*)

	(*ID Current Value*)
(*	anTool_Score					AT%I* 	: ARRAY [0..7] OF DINT;			*)

	(*ID Status*)
	bChange_Program_Ack 			AT%I*	: BOOL;							
	bChange_Program_Failed			AT%I*	: BOOL;							
(*	bResult_Valid_00				AT%I*	: BOOL;
	bTotal_Status_OK_00				AT%I*	: BOOL;

	bResult_Valid_01				AT%I*	: BOOL;
	bRegist_Master_Image_Ack		AT%I*	: BOOL;
	bRegist_Master_Image_Failed		AT%I*	: BOOL;							*)
	bTotal_Status_OK_01				AT%I*	: BOOL;
	bTotal_Status_NG				AT%I*	: BOOL;
(*	bError_status					AT%I*	: BOOL;
	bClear_Error_Ack				AT%I*	: BOOL;							*)
	bRun							AT%I*	: BOOL;
	bBusy							AT%I*	: BOOL;
	bTrigger_Ready					AT%I*	: BOOL;
	bTrigger_Ack					AT%I*	: BOOL;
(*	bTrigger_Failed					AT%I*	: BOOL;
	bResult_Updated_Toggle			AT%I*	: BOOL;
	bCount_Up_Ack					AT%I*	: BOOL;
	bReset_Statistics_Ack			AT%I*	: BOOL;
	bReset_Count_Ack				AT%I*	: BOOL;

	abTool_Invalid					AT%I* 	: ARRAY [0..6] OF BOOL;
	abTool_State					AT%I* 	: ARRAY [0..6] OF BOOL;			*)
	abProgram_Num					AT%I* 	: ARRAY [0..6] OF BOOL;			
(*	abLogic							AT%I* 	: ARRAY [0..4] OF BOOL;

	bSD_Card_Detected				AT%I*	: BOOL;
	bSD_Save_Stop_Ack				AT%I*	: BOOL;
	bSD_Card_No_Space				AT%I*	: BOOL;

	(*WcState*)
	bWcState						AT%I*	: BOOL;
	bInputToggle					AT%I*	: BOOL;							*)

	(*Info Data*)
	nState							AT%I*	: UINT;
(*	bAdsAddr						AT%I*	: ARRAY [0..5] OF USINT;		*)

END_VAR
(* Zeiten *)
fb_ton_quitt(IN:= , PT:= t#100ms, Q=> , ET=> );

(* Aufrufe *)
	Btn_Init();
	Control();
	ErrorHandling();

(* Toplevel *)
IF	sConfig.Aktiv THEN
	IF 	NOT Connected THEN
		sm_kamera_nicht_bb := TRUE;
		fb_state_entry.i16_next_step := FEHLER;
	END_IF
ELSE
	fb_state_entry.i16_next_step := INAKTIV;
END_IF

IF fb_state_entry.i16_next_step > INIT AND fb_state_entry.i16_next_step < FEHLER THEN
	IF fb_state_entry.i16_next_step < STOP THEN
		IF 	st_ctrl_in.b_stop THEN
			fb_state_entry.i16_next_step := STOP;
		END_IF
		IF 	bError_Status_00 THEN
			sm_kamera_controler_error := TRUE;
			fb_state_entry.i16_next_step := FEHLER;
		END_IF
	END_IF
END_IF

(* ==================================Schrittkette================================ *)
fb_state_entry(i16_pos:= 1);

CASE fb_state_entry.i16_step OF
(*=======================================================*)
INIT_OBJ:
	fb_state_entry.i16_next_step := INIT;

(*=======================================================*)
INIT:
	IF 	fb_state_entry.E THEN
		fb_ton_quitt.IN := FALSE;
		st_ctrl_out := st_ctrl_out_Empty;

		b_Kam_Pruef_IO := FALSE;
		b_Kam_Pruef_NIO := FALSE;
		sm_kamera_nicht_bb := FALSE;
		sm_kamera_keine_reaktion := FALSE;
		sm_jobnummer_nicht_erlaubt := FALSE;
		sm_kamera_controler_error := FALSE;
		Error.No:=0;
		Error.Text:='';
	END_IF

	(*-----------------------Weiterschaltbedingungen----------------------------*)
	IF st_ctrl_in.b_init THEN
		fb_state_entry.i16_next_step := 20;
	END_IF

(*=======================================================*)
20: fb_state_entry.s_debugtext:='Reset';

	stControl.bReset:=TRUE;

	IF 	fb_state_entry.fb_ton_Step.ET > t#100ms THEN
		fb_state_entry.i16_next_step := BEREIT;
	END_IF

	IF 	fb_state_entry.X THEN
		stControl.bReset:=FALSE;
	END_IF

(*=======================================================*)
BEREIT: fb_state_entry.s_debugtext:='waiting for start';

	IF 	fb_state_entry.E THEN
		st_ctrl_out.b_bereit := TRUE;
	END_IF

	(*-----------------------Weiterschaltbedingungen----------------------------*)
	IF	st_ctrl_in.b_start THEN
		b_Kam_Pruef_IO := FALSE;
		b_Kam_Pruef_NIO := FALSE;
		fb_state_entry.i16_next_step := 110;
	END_IF

	IF 	fb_state_entry.X THEN
		st_ctrl_out.b_busy := TRUE;
		st_ctrl_out.b_bereit := FALSE;
		st_ctrl_out.b_fertig := FALSE;
	END_IF

(*=======================================================*)
110: fb_state_entry.s_debugtext:='check job number';

	IF 	fb_state_entry.E THEN
		stControl.bReset:=TRUE;
	END_IF

	(*-----------------------Weiterschaltbedingungen----------------------------*)

	IF 	JobNo <> ActJobNo THEN
		IF 	bRun AND
			NOT bBusy AND
			NOT bChange_Program_Ack THEN
				fb_state_entry.i16_next_step:=120;
		END_IF
	ELSE
		fb_state_entry.i16_next_step := 140;
	END_IF

	IF 	fb_state_entry.X THEN
		stControl.bReset:=FALSE;
	END_IF

(*=======================================================*)
120: fb_state_entry.s_debugtext:='set job number';

	IF 	fb_state_entry.E THEN
		IF 	JobNo < 0 AND JobNo > 15 THEN
			sm_jobnummer_nicht_erlaubt := TRUE;
			fb_state_entry.i16_next_step := FEHLER;
		ELSE
			stControl.bPrgChange:=TRUE;
			stControl.iJobNo:= JobNo;
		END_IF
	END_IF

	(*-----------------------Weiterschaltbedingungen----------------------------*)
	IF 	bChange_Program_Ack THEN
		fb_state_entry.i16_next_step:=130;
	ELSIF fb_state_entry.fb_ton_Step.ET > t#5s THEN
		sm_kamera_keine_reaktion := TRUE;
		fb_state_entry.i16_next_step := FEHLER;
	END_IF


	IF 	fb_state_entry.X THEN
		stControl.bPrgChange:=FALSE;
		stControl.iJobNo:= 0;
	END_IF

(*=======================================================*)
130: fb_state_entry.s_debugtext:='check job number';

	IF 	JobNo = ActJobNo AND
		NOT bChange_Program_Failed THEN
		fb_state_entry.i16_next_step := 140;
	END_IF

(*=======================================================*)
140: fb_state_entry.s_debugtext:='Reset and check Ready';

	IF 	fb_state_entry.E THEN
		stControl.bReset:=TRUE;
	END_IF

	(*-----------------------Weiterschaltbedingungen----------------------------*)

	IF 	bRun AND
		NOT bBusy AND
		bTrigger_Ready THEN
		fb_state_entry.i16_next_step:=150;
	END_IF

	IF 	fb_state_entry.X THEN
		stControl.bReset:=FALSE;
	END_IF

(*=======================================================*)
150: fb_state_entry.s_debugtext:='set trigger';

	stControl.bTrigger :=TRUE;
	(*-----------------------Weiterschaltbedingungen----------------------------*)
	IF 	bTrigger_Ack THEN
		fb_state_entry.i16_next_step:=160;
	ELSIF fb_state_entry.fb_ton_Step.ET > t#5s THEN
		sm_kamera_keine_reaktion := TRUE;
		fb_state_entry.i16_next_step := FEHLER;
	END_IF

	IF 	fb_state_entry.X THEN
		stControl.bTrigger:=FALSE;
	END_IF

(*=======================================================*)
160: fb_state_entry.s_debugtext:='result of camera';

	IF 	NOT bBusy AND
		bTotal_Status_OK_01 <> bTotal_Status_NG THEN
		b_Kam_Pruef_IO 	:= bTotal_Status_OK_01;
		b_Kam_Pruef_NIO := bTotal_Status_NG;
		fb_state_entry.i16_next_step := BEREIT;
	ELSIF fb_state_entry.fb_ton_Step.ET > t#5s THEN
		sm_kamera_keine_reaktion := TRUE;
		fb_state_entry.i16_next_step := FEHLER;
	END_IF

	IF 	fb_state_entry.X THEN
		st_ctrl_out.b_busy:=FALSE;
		st_ctrl_out.b_fertig := TRUE;
	END_IF

(*=======================================================*)
STOP, FEHLER:

	IF 	fb_state_entry.E THEN
		st_ctrl_out := st_ctrl_out_Empty;
		st_ctrl_out.b_gestoppt := fb_state_entry.i16_next_step = STOP;
		st_ctrl_out.b_fehler := fb_state_entry.i16_next_step = FEHLER;
		fb_ton_quitt.IN := FALSE;
	END_IF

		IF	sm_kamera_keine_reaktion THEN
			FB_ReadXmlLineMsg.ID:='sm_kamera_keine_reaktion';
			Error.No:=1;
		ELSIF
			sm_kamera_nicht_bb THEN
			FB_ReadXmlLineMsg.ID:='sm_kamera_nicht_bb';
			Error.No:=2;
		ELSIF
			sm_jobnummer_nicht_erlaubt THEN
			FB_ReadXmlLineMsg.ID:='sm_jobnummer_nicht_erlaubt';
			Error.No:=3;
		ELSIF
			sm_kamera_controler_error THEN
			FB_ReadXmlLineMsg.ID:='sm_kamera_controler_error';
			Error.No:=4;
		END_IF

	(*-----------------------Weiterschaltbedingungen----------------------------*)
	IF 	st_ctrl_in.b_quitt OR gResetAll THEN
		fb_ton_quitt.IN := TRUE;
	END_IF

	IF 	fb_ton_quitt.Q THEN
		fb_ton_quitt.IN := FALSE;
		fb_state_entry.i16_next_step := INIT;
	END_IF

(*=======================================================*)
INAKTIV:

	IF 	fb_state_entry.E THEN
		st_ctrl_out := st_ctrl_out_Empty;
	END_IF
	st_ctrl_out.b_bereit := TRUE;
	(*-----------------------Weiterschaltbedingungen----------------------------*)
	IF	sConfig.Aktiv THEN
		fb_state_entry.i16_next_step := INIT;
	END_IF

END_CASE

fb_state_entry(i16_pos:= 2);
st_ctrl_in := st_ctrl_in_Empty;
END_FUNCTION_BLOCK
ACTION Btn_Init:
(*=====================================================================*)
BtnConnect.Text:='Connect';
BtnConnect.BackgroundColor:=Color.darkgrey;
BtnConnect.Enable:= TRUE; (*ModeSelect.Mode <> MODE_MANUAL;*)
IF	BtnConnect.Enable THEN
	BtnConnect.TextColor:=Color.grey;
ELSE
	BtnConnect.TextColor:=Color.black;
END_IF
BtnConnect.Visible:=TRUE;

(*=====================================================================*)
BtnTrigger.Text:='Trigger';
BtnTrigger.BackgroundColor:=Color.darkgrey;
BtnTrigger.Enable:= TRUE; (* ModeSelect.Mode <> MODE_MANUAL;*)
IF	BtnTrigger.Enable THEN
	BtnTrigger.TextColor:=Color.grey;
ELSE
	BtnTrigger.TextColor:=Color.black;
END_IF
BtnTrigger.Visible:=TRUE;
END_ACTION
ACTION Control:
(* DL-EC1A: PDO-Kommunikation (Prozessdaten-Objekte)*)
			Connected:= nState = 8; 								(* 0x0008 = Slave in 'OP' state *)

(* Index: 7000  SubIndex: 1 - 5 *)

FOR i := 0 TO 4 DO
(*Bit 0*) 	anInputRequest[i].0:=stControl.bReset;					(*Reserviert (alles zurücksetzen)*)
END_FOR

(*Bit 1*) 	anInputRequest[0].1:=stControl.bPrgChange;				(*Programmwechselanforderung*)
			anInputRequest[1].1:=stControl.iJobNo.0;
			anInputRequest[2].1:=stControl.iJobNo.1;
			anInputRequest[3].1:=stControl.iJobNo.2;
			anInputRequest[4].1:=stControl.iJobNo.3;

			ActJobNo.0:=abProgram_Num[0];
			ActJobNo.1:=abProgram_Num[1];
			ActJobNo.2:=abProgram_Num[2];
			ActJobNo.3:=abProgram_Num[3];

(*Bit 2*) 	anInputRequest[0].2:=stControl.bTrigger;				(*Trigger*)

(*nicht benutzt*)
(*Bit 3*) 	anInputRequest[0].3	:=stControl.bMaster;				(*Master-Registrierunganforderung *)
(*Bit 4*) 	anInputRequest[0].4	:=stControl.bSpeicherstopp;			(*Speicherstopp SD-Karte Anfrage*)
(*Bit 5*) 	anInputRequest[0].5	:=stControl.bStatistikruecksetzung;	(* Statistikrücksetzung anfordern*)
(*Bit 6*) 	anInputRequest[0].6	:=stControl.bFehlerLoeschen;		(*Anforderung Fehler löschen*)
(*Bit 7*) 	anInputRequest[0].7	:=stControl.OCR_Seriennummer;		(*Anforderung OCR-Seriennummer Hochzählen*)
(*Bit 8*) 	anInputRequest[0].8	:=stControl.Zaehlung_Ruecksetzen;	(*Zählung-Rücksetzen Anforderung*)
(*Bit 9*) 	anInputRequest[0].9	:=stControl.Statistik_Ruecksetzen;	(*Anforderung Statistik aller Programme Rücksetzen*)
(*Bit 10*) 	anInputRequest[0].10:=stControl.Reserviert_10;
(*Bit 11*) 	anInputRequest[0].11:=stControl.Reserviert_11;
(*Bit 12*) 	anInputRequest[0].12:=stControl.Reserviert_12;
(*Bit 13*) 	anInputRequest[0].13:=stControl.Reserviert_13;
(*Bit 14*) 	anInputRequest[0].14:=stControl.Reserviert_14;
(*Bit 15*) 	anInputRequest[0].15:=stControl.Reserviert_15;
END_ACTION
ACTION ErrorHandling:
(*------------------------------------------------------------------
	Error-Handling
  ------------------------------------------------------------------*)

FB_ReadXmlLineConf(
	Prefix:= 'CONFIG',
	ID:= sConfig.InstName,
	File:= 'CONFIG.xml',
	Text=>  );

FB_ReadXmlLineMsg(
	Prefix:= 'MSG',
	ID:= ,
	File:= 'MSG.xml',
	Text=>);

IF	NOT st_ctrl_out.b_fehler OR NOT sConfig.Aktiv THEN
	Error.No:=0;
	Error.Text:='';
	TempErrorText:='';
END_IF

IF 	Error.Text<>''	AND ST_Lng.b_EndChangeLng THEN
	Error.Typ:=0;
	ErrorHandler.AddError(ErrorToAdd:=Error,
						sVisu:=Visu.ErrorHandler);
END_IF

IF	 st_ctrl_out.b_fehler THEN
	Error.Text:=FB_ReadXmlLineConf.Text;
	Error.Text:=CONCAT(Error.Text,': ');
	Error.Text:=CONCAT(Error.Text,FB_ReadXmlLineMsg.Text);
END_IF
END_ACTION

(* POU zLibrary/Sensopart/FB_Sensopart, ST *)
FUNCTION_BLOCK FB_Sensopart
VAR_INPUT
	b_init							: BOOL;
	b_start							: BOOL;
	b_start_manual					: BOOL;
	b_quitt							: BOOL;
	b_reset							: BOOL;
	b_kamera_aktiv 					: BOOL;
	i16_job							: INT:=1;
	st_Description					: STRING;
END_VAR
VAR_OUTPUT
	b_ready							: BOOL;
	b_done							: BOOL;
	b_busy							: BOOL;
	b_error							: BOOL;

(* Ausgänge der Kamera *)
	Ergebnis_IO						: BOOL;
	Ergebnis_NIO					: BOOL;
	sm_kamera_nicht_bb				: BOOL := FALSE;
	sm_zeitueberschreitung			: BOOL := FALSE;
END_VAR
VAR
	b_first_cycle					: BOOL := TRUE;
	fb_ton_quitt					: TON;
	fb_ton_trigger					: TON;
	fb_tof_trigger					: TOF;
	fb_state_entry					: ST_StateEntry;
	fb_r_trig_start					: R_TRIG;
	fb_r_trig_trigger				: R_TRIG;
END_VAR

VAR_OUTPUT
	(*Sensopart Kamera*)
	a_Trigger 				AT %Q*: BOOL;
	a_Job_Bit1 				AT %Q*: BOOL;
	a_Job_Bit2 				AT %Q*: BOOL;
	a_Job_Bit3 				AT %Q*: BOOL;
	a_Job_Bit4 				AT %Q*: BOOL;
END_VAR
VAR

(* Eingänge von der Kamera *)
	e_Ergebnis_iO			AT %I*: BOOL;
	e_Ergebnis_niO			AT %I*: BOOL;
	e_Betriebsbereit		AT %I*: BOOL;
	e_Best_Jobwechsel		AT %I*: BOOL;
END_VAR
IF b_first_cycle THEN
	b_first_cycle := FALSE;
END_IF

a_Job_Bit1:=i16_job.0;
a_Job_Bit2:=i16_job.1;
a_Job_Bit3:=i16_job.2;
a_Job_Bit4:=i16_job.3;

(* Zeiten *)
fb_ton_quitt(IN:= , PT:= t#100ms, Q=> , ET=> );
fb_ton_trigger(IN:= , PT:= t#150ms, Q=> , ET=> );
fb_tof_trigger(IN:= fb_r_trig_trigger.Q , PT:= t#150ms, Q=> , ET=> );

(* Flanken *)
fb_r_trig_start(CLK:= b_start OR b_start_manual, Q=> );


IF	NOT b_kamera_aktiv THEN
	fb_state_entry.i16_next_step := INAKTIV;
END_IF

(* ==================================Schrittkette================================ *)
fb_state_entry(i16_pos:= 1);

CASE fb_state_entry.i16_step OF
(*=======================================================*)
	INIT_OBJ:
		fb_state_entry.i16_next_step := INIT;

(*=======================================================*)
	INIT:
		IF 	fb_state_entry.E THEN
			b_ready := FALSE;
			b_done := FALSE;
			b_quitt := FALSE;
			b_reset := FALSE;
			b_busy := FALSE;
			b_error := FALSE;
			b_start := FALSE;
			a_Trigger  := FALSE;
			Ergebnis_IO := FALSE;
			Ergebnis_NIO := FALSE;
			sm_kamera_nicht_bb := FALSE;
			sm_zeitueberschreitung := FALSE;
		END_IF

		(*-----------------------Weiterschaltbedingungen----------------------------*)
		IF 	b_init THEN
			IF  NOT b_kamera_aktiv THEN
				fb_state_entry.i16_next_step := BEREIT;		(* Kamera ist inaktiv *)
			ELSE
				fb_state_entry.i16_next_step := 20;			(* Kamera ist aktiv *)
			END_IF
		END_IF

(*=======================================================*)
	20: fb_state_entry.s_debugtext:='Kurze Wartezeit';

		IF 	fb_state_entry.fb_ton_Step.ET > t#300ms THEN
			fb_state_entry.i16_next_step := 30;
		END_IF

(*=======================================================*)
	30: fb_state_entry.s_debugtext:='Kamera Betriebsbereit';

		(*-----------------------Weiterschaltbedingungen----------------------------*)
		IF 	e_Betriebsbereit THEN
			fb_state_entry.i16_next_step := BEREIT;
		ELSIF
		 	fb_state_entry.fb_ton_Step.ET > t#300ms THEN
			sm_kamera_nicht_bb := TRUE;
			fb_state_entry.i16_next_step := FEHLER;
		END_IF

(*=======================================================*)
	BEREIT: fb_state_entry.s_debugtext:='warte auf Start';

		IF fb_state_entry.E THEN
			b_ready := TRUE;
			b_done := TRUE;
		END_IF

		(*-----------------------Weiterschaltbedingungen----------------------------*)
		IF 	b_kamera_aktiv THEN			(* Kamera aktiv *)
			IF 	fb_r_trig_start.Q AND e_Betriebsbereit THEN
				b_start := FALSE;
				b_busy := TRUE;
				b_done := FALSE;
				Ergebnis_IO := FALSE;
				Ergebnis_NIO := FALSE;
				fb_state_entry.i16_next_step := 102;
			ELSIF
				NOT e_Betriebsbereit THEN
				sm_kamera_nicht_bb := TRUE;
				fb_state_entry.i16_next_step := FEHLER;
			END_IF
		ELSE							(* Simulation der Kamera *)
			IF 	fb_r_trig_start.Q THEN
				b_busy := TRUE;
				b_done := FALSE;
				b_start:=FALSE;
				Ergebnis_IO := FALSE;
				Ergebnis_NIO := FALSE;
				fb_state_entry.i16_next_step := 300;
			END_IF
		END_IF

(*=======================================================*)
	102: fb_state_entry.s_debugtext:='Jobwechsel';

		IF 	fb_state_entry.fb_ton_Step.ET > t#1s OR
			e_Best_Jobwechsel THEN
			fb_state_entry.i16_next_step := 105;
		END_IF

(*=======================================================*)
	105: fb_state_entry.s_debugtext:='Kamera wieder bereit';

		IF 	e_Betriebsbereit THEN
			fb_state_entry.i16_next_step := 110;
		ELSIF
			NOT e_Betriebsbereit AND fb_state_entry.fb_ton_Step.ET > t#2s THEN
			sm_kamera_nicht_bb := TRUE;
			fb_state_entry.i16_next_step := FEHLER;
		END_IF

(*=======================================================*)
	110: fb_state_entry.s_debugtext:='Trigger setzen ';

		IF 	fb_state_entry.E THEN
			a_Trigger := TRUE;
			Ergebnis_IO := FALSE;
			Ergebnis_NIO := FALSE;
			fb_ton_trigger.IN := TRUE;
		END_IF

		(*-----------------------Weiterschaltbedingungen----------------------------*)
		IF 	fb_ton_trigger.Q THEN
			a_Trigger := FALSE;
			fb_ton_trigger.IN := FALSE;
			fb_state_entry.i16_next_step := 130;
		END_IF

(*=======================================================*)
	120: fb_state_entry.s_debugtext:='Warten auf Ergebnis der Kamera';

		IF 	NOT e_Ergebnis_iO AND
			NOT e_Ergebnis_niO THEN
			fb_state_entry.i16_next_step := 130;
		ELSIF
			fb_state_entry.fb_ton_Step.ET > t#4000ms THEN
			sm_zeitueberschreitung := TRUE;
			fb_state_entry.i16_next_step := FEHLER;
		END_IF

(*=======================================================*)
	130: fb_state_entry.s_debugtext:='Warten auf Ergebnis der Kamera ';

		IF 	NOT fb_state_entry.E AND e_Ergebnis_iO AND e_Betriebsbereit THEN
			Ergebnis_IO := TRUE;
			fb_state_entry.i16_next_step := BEREIT;
		ELSIF
			NOT fb_state_entry.E AND e_Ergebnis_niO AND e_Betriebsbereit THEN
			Ergebnis_NIO := TRUE;
			fb_state_entry.i16_next_step := BEREIT;
		ELSIF
			fb_state_entry.fb_ton_Step.ET > t#4000ms THEN
			sm_zeitueberschreitung := TRUE;
			fb_state_entry.i16_next_step := FEHLER;
		END_IF

		IF 	fb_state_entry.X THEN
			b_busy := FALSE;
			b_done := TRUE;
		END_IF

(*=======================================================*)
	300: fb_state_entry.s_debugtext:='Kamera ist nicht aktiv (Warten) ';		

		IF 	fb_state_entry.fb_ton_Step.ET > t#500ms THEN
			b_busy := FALSE;
			b_done := TRUE;
			Ergebnis_IO := TRUE;
			fb_state_entry.i16_next_step := BEREIT;
		END_IF

(*=======================================================*)
	STOP, FEHLER:
		IF 	fb_state_entry.E THEN
			b_error := TRUE;
			fb_ton_quitt.IN := FALSE;
			a_Trigger := FALSE;
		END_IF

		(*-----------------------Weiterschaltbedingungen----------------------------*)
		IF	(b_reset OR b_quitt) AND
			NOT fb_state_entry.E THEN
			b_error := FALSE;
			fb_ton_quitt.IN := TRUE;
		END_IF

		IF 	fb_ton_quitt.Q THEN
			fb_ton_quitt.IN := FALSE;
			fb_state_entry.i16_next_step := INIT;
		END_IF

(*=======================================================*)
	INAKTIV:
		IF 	fb_state_entry.E THEN
			b_ready := FALSE;
			b_done := FALSE;
			b_busy := FALSE;
			b_start := FALSE;
		END_IF

		IF	b_kamera_aktiv THEN
			fb_state_entry.i16_next_step := STOP;
		END_IF

END_CASE

fb_state_entry(i16_pos:= 2);
END_FUNCTION_BLOCK

(* POU zLibrary/Sensopart/FB_SensopartEthernet, ST *)
FUNCTION_BLOCK FB_SensopartEthernet
VAR_INPUT
	Activated				: BOOL;
	JobNo					: INT;
	s_IpAdress				: STRING;
	i_DataPort				: UDINT;
	i_CmdPort				: UDINT;
	st_ctrl_in				: struct_ctrl_in;
	st_Description			: STRING;
	st_InstName				: STRING;
	SensopartErgebnis		: STRING(15); (*Ergebnis Sensopart Kamera*)
END_VAR
VAR_IN_OUT

END_VAR
VAR_OUTPUT
	st_ctrl_out				: struct_ctrl_out;
	Connected				: BOOL;							(* Sockets Connected*)
	RecvDataString			: T_MaxString;
	ActJobNo				: INT;
END_VAR
VAR
	fb_ton_quitt						: TON;
	fb_state_entry					: ST_StateEntry;
	fb_state_entry_command			: ST_StateEntry;

	(* Error Handling *)
	FB_ReadXmlLineConf			: FB_ReadXmlLine;
	FB_ReadXmlLineMsg			: FB_ReadXmlLine;
	(*Variablen für Behr Meldungen*)
	TempErrorText					: STRING(255);
	ProcessTime					: DINT;				(* Counts the time in steps of 100ms since starting operation *)
	Error							: ErrorStruct;

	sm_kamera_keine_reaktion		: BOOL;
	sm_kamera_nicht_bb			: BOOL;
	sm_jobnummer_nicht_erlaubt		: BOOL;		(* erlaubter Bereich von 1-255 *)
	sm_kamera_command_error		: BOOL;
	sm_kamera_connect_error		: BOOL;
	sm_kamera_send_error			: BOOL;
	sm_kamera_rec_error			: BOOL;

	(*TcpIp-Connection via Socket*)
	FBClientServerConnectionCmd 	: FB_ClientServerConnection;
	FBClientServerConnectionRcv 	: FB_ClientServerConnection;
	FBSocketSend					: FB_SocketSend;
	FBSocketRecv					: FB_SocketReceive;
	SocketHandleCmd				: T_HSOCKET;
	SocketHandleRcv				: T_HSOCKET;
	ErrorId						: UDINT;
	nRecBytes					: UDINT;						(* Contains the number of bytes currently received. *)

	RecvStringCmd				: STRING(25);

	TRG_CMD:		ARRAY [0..2] OF BYTE:= 16#54,16#52,16#47;	(* [T, R, G] Trigger *)
	CJB_CMD:		ARRAY [0..5] OF BYTE:= 16#43,16#4A,16#42;	(* [C, J, B, 0, 0, 1] ChangeJoB z.B für Jobnummer 1 *)
	CJB_RCV:		ARRAY [0..7] OF BYTE;

	JbNoMem					: INT;
	CalcJbNo					: BYTE;

	b_Kam_Pruef_IO			:BOOL; 				(* Kameraprüfung Ergebnis iO *)
	b_Kam_Pruef_NIO			:BOOL; 				(* Kameraprüfung Ergebnis niO *)

	b_Kam_Bereit	  			: BOOL;				(* Bereit für nächsten ext. Trigger *)
	b_Betriebsbereit_eth			: BOOL:=FALSE;	(* Bereit kommt von EtherNet (noch nicht programmiert) *)
	e_Betriebsbereit  		AT %I*: BOOL;			(* Bereit kommt nur über Hardware-Eingang *)
 	BtnConnect					: sButtonVisu;
	BtnTrigger					: sButtonVisu;

END_VAR
(* Zeiten *)
fb_ton_quitt(IN:= , PT:= t#100ms, Q=> , ET=> );

(* Aufrufe *)
Btn_Init();
Command();
ErrorHandling();

b_Kam_Bereit := e_Betriebsbereit OR b_Betriebsbereit_eth;	(* Betriebsbereit  von EtherNet oder Eingang *)

(* Toplevel *)
IF	NOT Activated THEN
	fb_state_entry.i16_next_step := INAKTIV;
END_IF

IF fb_state_entry.i16_next_step > INIT AND fb_state_entry.i16_next_step < FEHLER THEN
	IF fb_state_entry.i16_next_step < STOP THEN
		IF st_ctrl_in.b_stop THEN
			fb_state_entry.i16_next_step := STOP;
		END_IF
		IF 	sm_kamera_command_error OR
			sm_kamera_send_error OR
			sm_kamera_rec_error OR
			sm_kamera_connect_error THEN
			fb_state_entry.i16_next_step := FEHLER;
		END_IF
	END_IF
END_IF

(* ==================================Schrittkette================================ *)
fb_state_entry(i16_pos:= 1);

CASE fb_state_entry.i16_step OF
(*=======================================================*)
INIT_OBJ:

	fb_state_entry.i16_next_step := INIT;

(*=======================================================*)
INIT:
	IF 	fb_state_entry.E THEN
		fb_ton_quitt.IN := FALSE;
		st_ctrl_out := st_ctrl_out_Empty;
		b_Kam_Pruef_IO := FALSE;
		b_Kam_Pruef_NIO := FALSE;
		sm_kamera_nicht_bb := FALSE;
		sm_kamera_keine_reaktion := FALSE;
		sm_jobnummer_nicht_erlaubt := FALSE;
		sm_kamera_command_error:=FALSE;
		sm_kamera_connect_error:=FALSE;
		sm_kamera_send_error:=FALSE;
		sm_kamera_rec_error:=FALSE;
		Error.No:=0;
		Error.Text:='';
	END_IF

	(*-----------------------Weiterschaltbedingungen----------------------------*)
	IF	BtnConnect.tasten OR
		st_ctrl_in.b_init THEN
		fb_state_entry.i16_next_step := 30;
	END_IF

(*=======================================================*)
30: fb_state_entry.s_debugtext:='start Connect';

	IF	fb_state_entry.E THEN
		fb_state_entry_command.i16_next_step:=20;
	END_IF

	(*-----------------------Weiterschaltbedingungen----------------------------*)
	IF 	fb_state_entry_command.i16_step > INIT THEN
		fb_state_entry.i16_next_step := 35;
	ELSIF
		fb_state_entry.fb_ton_Step.ET > t#2s THEN
		sm_kamera_nicht_bb := TRUE;
		fb_state_entry.i16_next_step := FEHLER;
	END_IF

(*=======================================================*)
35: fb_state_entry.s_debugtext:='warte auf bereit von connect';

	IF 	fb_state_entry_command.i16_step = BEREIT THEN
		fb_state_entry.i16_next_step := BEREIT;
	ELSIF
		fb_state_entry.fb_ton_Step.ET > t#20s THEN
		sm_kamera_nicht_bb := TRUE;
		fb_state_entry.i16_next_step := FEHLER;
	END_IF

(*=======================================================*)
BEREIT: fb_state_entry.s_debugtext:='warte auf Start';

	IF 	fb_state_entry.E THEN
		st_ctrl_out.b_bereit := TRUE;
		st_ctrl_in.b_start:=FALSE;
	END_IF

	(*-----------------------Weiterschaltbedingungen----------------------------*)
	IF 	(b_Kam_Bereit OR NOT Activated) AND
		(st_ctrl_in.b_start OR BtnTrigger.tasten) THEN
		b_Kam_Pruef_IO := FALSE;
		b_Kam_Pruef_NIO := FALSE;
		fb_state_entry.i16_next_step := 110;
	ELSIF
		fb_state_entry.fb_ton_Step.ET > t#1s AND
		(NOT b_Kam_Bereit OR NOT Connected) AND
		Activated THEN
		sm_kamera_nicht_bb := TRUE;
		fb_state_entry.i16_next_step := FEHLER;
	END_IF

	IF 	fb_state_entry.X THEN
		st_ctrl_out.b_busy:=TRUE;
		st_ctrl_out.b_bereit := FALSE;
		st_ctrl_out.b_fertig := FALSE;
	END_IF

(*=======================================================*)
110: fb_state_entry.s_debugtext:='Jobnummer im erlaubten Bereich?';

	(*-----------------------Weiterschaltbedingungen----------------------------*)
	IF 	JobNo > 0 AND
		JobNo < 256 THEN
		fb_state_entry.i16_next_step := 120;
	ELSE
		sm_jobnummer_nicht_erlaubt := TRUE;
		fb_state_entry.i16_next_step := FEHLER;
	END_IF

(*=======================================================*)
120: fb_state_entry.s_debugtext:='Trigger setzen';

	IF 	fb_state_entry.E THEN
		fb_state_entry_command.i16_next_step:=110;
		b_Kam_Pruef_IO := FALSE;
		b_Kam_Pruef_NIO := FALSE;
	END_IF

	(*-----------------------Weiterschaltbedingungen----------------------------*)
	IF 	fb_state_entry_command.i16_step > BEREIT THEN
		fb_state_entry.i16_next_step := 130;
	ELSIF
		fb_state_entry.fb_ton_Step.ET > t#3s THEN
		sm_kamera_keine_reaktion := TRUE;
		fb_state_entry.i16_next_step := FEHLER;
	END_IF

(*=======================================================*)
130: fb_state_entry.s_debugtext:='warte bis Kamera fertig ist';

	(*-----------------------Weiterschaltbedingungen----------------------------*)
	IF 	fb_state_entry_command.i16_step = BEREIT THEN
		fb_state_entry.i16_next_step := 140;
	ELSIF
		fb_state_entry.fb_ton_Step.ET > t#5s THEN
		sm_kamera_keine_reaktion := TRUE;
		fb_state_entry.i16_next_step := FEHLER;
	END_IF

(*=======================================================*)
140: fb_state_entry.s_debugtext:='Ergebnis der Kamera auswerten';

	(*-----------------------Weiterschaltbedingungen----------------------------*)
	(*// RecvDataString Erklärung
	// 2 = Anzahl der Ausgangsbits der Kamera
	// P = Positives Ergebnis
	// F = Negatives Ergebnis
	// Jobnummer
	// evtl. Jobnummer anders abfragen*)
	IF 	RecvDataString = CONCAT(SensopartErgebnis, INT_TO_STRING(JobNo)) THEN		(* Stecker iO *)
		b_Kam_Pruef_IO :=  TRUE;
		fb_state_entry.i16_next_step := BEREIT;
	ELSE		(* Stecker niO *)
		b_Kam_Pruef_NIO :=  TRUE;
		fb_state_entry.i16_next_step := BEREIT;
	END_IF

	IF 	fb_state_entry.X THEN
		st_ctrl_out.b_busy:=FALSE;
		st_ctrl_out.b_fertig := TRUE;
	END_IF

(*=======================================================*)
STOP, FEHLER:

	IF 	fb_state_entry.E THEN
		st_ctrl_out := st_ctrl_out_Empty;
		st_ctrl_out.b_gestoppt := fb_state_entry.i16_next_step = STOP;
		st_ctrl_out.b_fehler := fb_state_entry.i16_next_step = FEHLER;
		fb_state_entry_command.i16_next_step:= fb_state_entry.i16_next_step;
		fb_ton_quitt.IN := FALSE;
	END_IF

	IF	sm_kamera_keine_reaktion THEN
		FB_ReadXmlLineMsg.ID:='sm_kamera_keine_reaktion';
		Error.No:=1;
	ELSIF
		sm_kamera_nicht_bb THEN
		FB_ReadXmlLineMsg.ID:='sm_kamera_nicht_bb';
		Error.No:=2;
	ELSIF
		sm_jobnummer_nicht_erlaubt THEN
		FB_ReadXmlLineMsg.ID:='sm_jobnummer_nicht_erlaubt';
		Error.No:=3;
	ELSIF
		sm_kamera_command_error THEN
		FB_ReadXmlLineMsg.ID:='sm_kamera_command_error';
		Error.No:=4;
	ELSIF
		sm_kamera_connect_error THEN
		FB_ReadXmlLineMsg.ID:='sm_kamera_connect_error';
		Error.No:=5;
	ELSIF
		sm_kamera_send_error THEN
		FB_ReadXmlLineMsg.ID:='sm_kamera_send_error';
		Error.No:=6;
	ELSIF
		sm_kamera_rec_error THEN
		FB_ReadXmlLineMsg.ID:='sm_kamera_rec_error';
		Error.No:=7;
	END_IF

	(*-----------------------Weiterschaltbedingungen----------------------------*)
	IF 	(st_ctrl_in.b_quitt OR gResetAll) THEN
		fb_ton_quitt.IN := TRUE;
	END_IF

	IF 	fb_ton_quitt.Q THEN
		fb_ton_quitt.IN := FALSE;
		fb_state_entry.i16_next_step := INIT;
	END_IF

(*=======================================================*)
INAKTIV:

	IF 	fb_state_entry.E THEN
		st_ctrl_out := st_ctrl_out_Empty;
	END_IF

	st_ctrl_out.b_bereit := TRUE;
	IF	Activated THEN
		fb_state_entry.i16_next_step := INIT;
	END_IF

END_CASE

fb_state_entry(i16_pos:= 2);
st_ctrl_in := st_ctrl_in_Empty;
END_FUNCTION_BLOCK
ACTION Btn_Init:
(*=====================================================================*)
BtnConnect.Text:='Connect';
BtnConnect.BackgroundColor:=Color.darkgrey;
BtnConnect.Enable:= TRUE; (*ModeSelect.Mode <> MODE_MANUAL;*)
IF	BtnConnect.Enable THEN
	BtnConnect.TextColor:=Color.grey;
ELSE
	BtnConnect.TextColor:=Color.black;
END_IF
BtnConnect.Visible:=TRUE;

(*=====================================================================*)
BtnTrigger.Text:='Trigger';
BtnTrigger.BackgroundColor:=Color.darkgrey;
BtnTrigger.Enable:= TRUE; (* ModeSelect.Mode <> MODE_MANUAL;*)
IF	BtnTrigger.Enable THEN
	BtnTrigger.TextColor:=Color.grey;
ELSE
	BtnTrigger.TextColor:=Color.black;
END_IF
BtnTrigger.Visible:=TRUE;
END_ACTION
ACTION Command:
(*TemplateClass01_Function01: write here a short Description of this command*)

Connected:=	FBClientServerConnectionCmd.eState=eSOCKET_CONNECTED AND
				FBClientServerConnectionRcv.eState=eSOCKET_CONNECTED;

(* ==================================Schrittkette================================ *)
fb_state_entry_command(i16_pos:= 1);

CASE fb_state_entry_command.i16_step OF

INIT_OBJ:

	fb_state_entry_command.i16_next_step:=INIT;

(*===========================================================*)
INIT: fb_state_entry_command.s_debugtext:= 'INIT kommt vom Hauptablauf';

(*===========================================================*)
20:	fb_state_entry_command.s_debugtext:='Preset local Vars';

	FBClientServerConnectionCmd(bEnable:=FALSE);
	FBClientServerConnectionRcv(bEnable:=FALSE);
	FBSocketSend(bExecute:=FALSE);
	FBSocketRecv(bExecute:=FALSE);
	fb_state_entry_command.i16_next_step:=30;

(*===========================================================*)
30:	fb_state_entry_command.s_debugtext:='Create new Socket-Connection: Start';

	FBClientServerConnectionCmd
		(bEnable		:=TRUE,
		nMode			:=CONNECT_MODE_ENABLEDBG,	(* Enable Debugging (to see in SystemManager Logger*)
		sRemoteHost	:=s_IpAdress,						(* IP-Adresse NewPort-Achsregler *)
		nRemotePort	:=i_CmdPort,						(* TCPIP Socket Port *)
		tReconnect		:= t#10s);
	IF 	FBClientServerConnectionCmd.bBusy THEN
		fb_state_entry_command.i16_next_step:=40;
	END_IF

(*===========================================================*)
40:	fb_state_entry_command.s_debugtext:='Create new Socket-Connection: Finished';

	FBClientServerConnectionCmd
		(bEnable		:=TRUE,
		nMode			:=CONNECT_MODE_ENABLEDBG,	(* Enable Debugging (to see in SystemManager Logger*)
		sRemoteHost	:=s_IpAdress,						(* IP-Adresse NewPort-Achsregler *)
		nRemotePort	:=i_CmdPort,						(* TCPIP Socket Port *)
		tReconnect		:= t#10s);
	IF 	NOT FBClientServerConnectionCmd.bBusy AND
		NOT FBClientServerConnectionCmd.bError THEN
		SocketHandleCmd:=FBClientServerConnectionCmd.hSocket;
		fb_state_entry_command.i16_next_step:=50;
	ELSIF
		FBClientServerConnectionCmd.bError THEN
		sm_kamera_connect_error:=TRUE;
		fb_state_entry_command.i16_next_step:=FEHLER;
		ErrorId:=FBClientServerConnectionCmd.nErrId;
	END_IF

(*===========================================================*)
50:	fb_state_entry_command.s_debugtext:='Create new Socket-Connection: Start';

	FBClientServerConnectionRcv
		(bEnable		:=TRUE,
		nMode			:=CONNECT_MODE_ENABLEDBG,	(* Enable Debugging (to see in SystemManager Logger*)
		sRemoteHost	:=s_IpAdress,						(* IP-Adresse NewPort-Achsregler *)
		nRemotePort	:=i_DataPort,						(* TCPIP Socket Port *)
		tReconnect		:= t#10s);
	IF 	FBClientServerConnectionRcv.bBusy THEN
		fb_state_entry_command.i16_next_step:=60;
	END_IF

(*===========================================================*)
60:	fb_state_entry_command.s_debugtext:='Create new Socket-Connection: Finished';

	FBClientServerConnectionRcv
		(bEnable		:=TRUE,
		nMode			:=CONNECT_MODE_ENABLEDBG,	(* Enable Debugging (to see in SystemManager Logger*)
		sRemoteHost	:=s_IpAdress,						(* IP-Adresse NewPort-Achsregler *)
		nRemotePort	:=i_DataPort,						(* TCPIP Socket Port *)
		tReconnect		:= t#10s);
	IF 	NOT FBClientServerConnectionRcv.bBusy AND
		NOT FBClientServerConnectionRcv.bError THEN
		SocketHandleRcv:=FBClientServerConnectionRcv.hSocket;
		fb_state_entry_command.i16_next_step:=70;
	ELSIF
		FBClientServerConnectionRcv.bError THEN
		sm_kamera_connect_error:=TRUE;
		fb_state_entry_command.i16_next_step:=FEHLER;
		ErrorId:=FBClientServerConnectionRcv.nErrId;
	END_IF

(*===========================================================*)
70:	fb_state_entry_command.s_debugtext:='Check if Socket is correct connected';

	IF 	Connected AND
		SocketHandleCmd.handle>0 AND
		SocketHandleRcv.handle>0 THEN
		fb_state_entry_command.i16_next_step:=BEREIT;
	END_IF

(*=======================================================*)
BEREIT: fb_state_entry_command.s_debugtext:= 'START kommt vom Hauptablauf';

(*===========================================================*)
110: fb_state_entry_command.s_debugtext:='Check if Socket is correct connected';

	IF 	Connected AND
		SocketHandleCmd.handle>0 AND
		SocketHandleRcv.handle>0 AND
		b_Kam_Bereit AND
		Activated THEN
		IF 	JobNo=0 THEN
		 	 fb_state_entry_command.i16_next_step:=FEHLER;
		ELSE
			MEMSET(destAddr:=ADR(RecvDataString), fillByte:=0, n:=SIZEOF(RecvDataString));
			MEMSET(destAddr:=ADR(CJB_RCV), fillByte:=0, n:=SIZEOF(CJB_RCV));
			MEMSET(destAddr:=ADR(RecvStringCmd), fillByte:=0, n:=SIZEOF(RecvStringCmd));
			fb_state_entry_command.i16_next_step:=120;
		END_IF
	ELSE
		sm_kamera_connect_error:=TRUE;
		fb_state_entry_command.i16_next_step:=FEHLER;
	END_IF

(*===========================================================*)
120: fb_state_entry_command.s_debugtext:='Job-Nummer prüfen und setzen.';

	 IF 	JobNo <> ActJobNo THEN
		JbNoMem:=JobNo;
		CalcJbNo:=INT_TO_BYTE(JbNoMem/100);
		CJB_CMD[3]:=16#30+CalcJbNo;

		CalcJbNo:=CalcJbNo*100;
		JbNoMem:=JbNoMem-CalcJbNo;
		CalcJbNo:=INT_TO_BYTE(JbNoMem/10);
		CJB_CMD[4]:=16#30+CalcJbNo;

		CalcJbNo:=CalcJbNo*10;
		JbNoMem:=INT_TO_BYTE(JbNoMem-CalcJbNo);
		CJB_CMD[5]:=16#30+INT_TO_BYTE(JbNoMem);

		fb_state_entry_command.i16_next_step:=130;
	ELSE
		fb_state_entry_command.i16_next_step:=200;
	END_IF

(*===========================================================*)
130: fb_state_entry_command.s_debugtext:='start FBSocketSend';

	FBSocketSend(bExecute	:=TRUE,
				hSocket		:= SocketHandleCmd,
				cbLen			:= 6,
				pSrc			:= ADR(CJB_CMD),
				tTimeout		:= t#5s);
	IF 	FBSocketSend.bBusy THEN
		fb_state_entry_command.i16_next_step:=140;
	END_IF

(*===========================================================*)
140: fb_state_entry_command.s_debugtext:='warte auf fertig  FBSocketSend';

	FBSocketSend(bExecute:=FALSE);
	IF 	NOT FBSocketSend.bBusy AND
		NOT FBSocketSend.bError THEN
		fb_state_entry_command.i16_next_step:=150;
	ELSIF
		FBSocketSend.bError THEN
		sm_kamera_send_error:=TRUE;
		fb_state_entry_command.i16_next_step:=FEHLER;
		ErrorId:=FBSocketSend.nErrId;
	END_IF

(*===========================================================*)
150: fb_state_entry_command.s_debugtext:='Wait before Receive';

	IF 	fb_state_entry_command.fb_ton_Step.ET > T#0ms THEN
		fb_state_entry_command.i16_next_step:=160;
	END_IF

(*===========================================================*)
160: fb_state_entry_command.s_debugtext:='Receive starten';

	FBSocketRecv(	bExecute	:=TRUE,
					hSocket	:= SocketHandleCmd,
					cbLen		:= SIZEOF(CJB_RCV),
					pDest		:= ADR(CJB_RCV),
					tTimeout	:= t#5s );
	IF 	FBSocketRecv.bBusy THEN
		fb_state_entry_command.i16_next_step:=170;
	END_IF

(*===========================================================*)
170: fb_state_entry_command.s_debugtext:='Job-Nr. rücklesen';

	FBSocketRecv(bExecute:=FALSE);
	IF 	NOT FBSocketRecv.bBusy AND
		NOT FBSocketRecv.bError THEN
		nRecBytes:=FBSocketRecv.nRecBytes;
		fb_state_entry_command.i16_next_step:=180;
	ELSIF
		FBSocketRecv.bError THEN
		sm_kamera_rec_error:=TRUE;
		fb_state_entry_command.i16_next_step:=FEHLER;
		ErrorId:=FBSocketRecv.nErrId;
	END_IF

(*===========================================================*)
180: fb_state_entry_command.s_debugtext:='Empfangene Daten gültig';

	IF 	nRecBytes>0 THEN
		fb_state_entry_command.i16_next_step:=190;
	ELSE
		fb_state_entry_command.i16_next_step:=160;
	END_IF

(*===========================================================*)
190: fb_state_entry_command.s_debugtext:='prüfe Ergebniss';

	IF 	CJB_RCV[3] < 16#50 THEN
		ErrorId:=16#0040;
		sm_kamera_rec_error:=TRUE;
		fb_state_entry_command.i16_next_step:=FEHLER;
	ELSIF
		CJB_RCV[5] <> CJB_CMD[3] OR
		CJB_RCV[6] <> CJB_CMD[4] OR
		CJB_RCV[7] <> CJB_CMD[5] THEN
		ErrorId:=16#0050;
		sm_kamera_rec_error:=TRUE;
		fb_state_entry_command.i16_next_step:=FEHLER;
	ELSE
		ErrorId:=16#0000;
		ActJobNo:=(CJB_RCV[5]-16#30)*100+(CJB_RCV[6]-16#30)*10+(CJB_RCV[7]-16#30);
	 	fb_state_entry_command.i16_next_step:=200;
	END_IF

(*===========================================================*)
(*===========================================================*)
200: fb_state_entry_command.s_debugtext:='Trigger-Cmd senden';

	FBSocketSend(bExecute	:=TRUE,
				hSocket		:= SocketHandleCmd,
				cbLen			:= 3,
				pSrc			:= ADR(TRG_CMD),
				tTimeout		:= T#5S);
	IF 	FBSocketSend.bBusy THEN
		fb_state_entry_command.i16_next_step:=210;
	END_IF

(*===========================================================*)
210: fb_state_entry_command.s_debugtext:='warte auf fertig Trigger-Cmd';

	FBSocketSend(bExecute:=FALSE);
	IF 	NOT FBSocketSend.bBusy AND
		NOT FBSocketSend.bError THEN
		fb_state_entry_command.i16_next_step:=220;
	ELSIF
		FBSocketSend.bError THEN
		sm_kamera_send_error:=TRUE;
		fb_state_entry_command.i16_next_step:=FEHLER;
		ErrorId:=FBSocketSend.nErrId;
	END_IF

(*===========================================================*)
220: fb_state_entry_command.s_debugtext:='Wait before Receive';

	IF 	fb_state_entry_command.fb_ton_Step.ET > t#10ms THEN
		fb_state_entry_command.i16_next_step:=230;
	END_IF

(*===========================================================*)
230: fb_state_entry_command.s_debugtext:='Receive starten';

	FBSocketRecv(	bExecute	:=TRUE,
					hSocket	:= SocketHandleCmd,
					cbLen		:= SIZEOF(RecvStringCmd),
					pDest		:= ADR(RecvStringCmd),
					tTimeout	:= t#5s );
	IF 	FBSocketRecv.bBusy THEN
		fb_state_entry_command.i16_next_step:=240;
	END_IF

(*===========================================================*)
240: fb_state_entry_command.s_debugtext:='Receive-Buffer lesen';

	FBSocketRecv(bExecute:=FALSE);
	IF 	NOT FBSocketRecv.bBusy AND
		NOT FBSocketRecv.bError THEN
		nRecBytes:=FBSocketRecv.nRecBytes;
		fb_state_entry_command.i16_next_step:=250;
	ELSIF
		FBSocketRecv.bError THEN
		sm_kamera_rec_error:=TRUE;
		fb_state_entry_command.i16_next_step:=FEHLER;
		ErrorId:=FBSocketRecv.nErrId;
	END_IF

(*===========================================================*)
250: fb_state_entry_command.s_debugtext:='Response erhalten?';

	IF 	nRecBytes>0 THEN
		fb_state_entry_command.i16_next_step:=300;
	ELSE
		fb_state_entry_command.i16_next_step:=230;		(*wdh. bis etwas ankommt*)
	END_IF

(*===========================================================*)
(*===========================================================*)
300: fb_state_entry_command.s_debugtext:='Ergebnis-Daten von Datenport lesen';

	IF 	Activated THEN
		fb_state_entry_command.i16_next_step:=310;
	ELSE
		fb_state_entry_command.i16_next_step:=BEREIT;
	END_IF

(*===========================================================*)
310: fb_state_entry_command.s_debugtext:='Receive starten';

	FBSocketRecv(bExecute	:=TRUE,
				hSocket		:= SocketHandleRcv,
				cbLen			:= SIZEOF(RecvDataString),
				pDest			:= ADR(RecvDataString),
				tTimeout		:= T#5S );
	IF 	FBSocketRecv.bBusy THEN
		fb_state_entry_command.i16_next_step:=320;
	END_IF

(*===========================================================*)
320: fb_state_entry_command.s_debugtext:='Receive-Buffer lesen';

	FBSocketRecv(bExecute:=FALSE);
	IF 	NOT FBSocketRecv.bBusy AND
		NOT FBSocketRecv.bError THEN
		nRecBytes:=FBSocketRecv.nRecBytes;
		fb_state_entry_command.i16_next_step:=330;
	ELSIF
		FBSocketRecv.bError THEN
		sm_kamera_rec_error:=TRUE;
		fb_state_entry_command.i16_next_step:=FEHLER;
		ErrorId:=FBSocketRecv.nErrId;
	END_IF

(*===========================================================*)
330: fb_state_entry_command.s_debugtext:='Antwort erhalten?';

	IF 	nRecBytes>0 THEN
		fb_state_entry_command.i16_next_step:=BEREIT;
	ELSE
		fb_state_entry_command.i16_next_step:=310;		(*wdh. bis etwas ankommt*)
	END_IF

(*=======================================================*)
STOP, FEHLER:

	IF 	fb_ton_quitt.Q THEN
		fb_state_entry_command.i16_next_step := INIT;
	END_IF

END_CASE

fb_state_entry_command(i16_pos:= 2);
END_ACTION
ACTION ErrorHandling:
(*------------------------------------------------------------------
	Error-Handling
  ------------------------------------------------------------------*)

FB_ReadXmlLineConf(
	Prefix:= 'CONFIG',
	ID:= st_InstName,
	File:= 'CONFIG.xml',
	Text=>  );

FB_ReadXmlLineMsg(
	Prefix:= 'MSG',
	ID:= ,
	File:= 'MSG.xml',
	Text=>);

IF	NOT st_ctrl_out.b_fehler THEN	(*OR NOT Activated *)
	Error.No:=0;
	Error.Text:='';
	TempErrorText:='';
END_IF

IF 	Error.Text<>''	AND ST_Lng.b_EndChangeLng THEN
	Error.Typ:=0;
	ErrorHandler.AddError(ErrorToAdd:=Error,
						sVisu:=Visu.ErrorHandler);
END_IF

IF	 st_ctrl_out.b_fehler THEN
	Error.Text:=FB_ReadXmlLineConf.Text;
	Error.Text:=CONCAT(Error.Text,': ');
	Error.Text:=CONCAT(Error.Text,FB_ReadXmlLineMsg.Text);
END_IF
END_ACTION

(* Visualisation MAIN
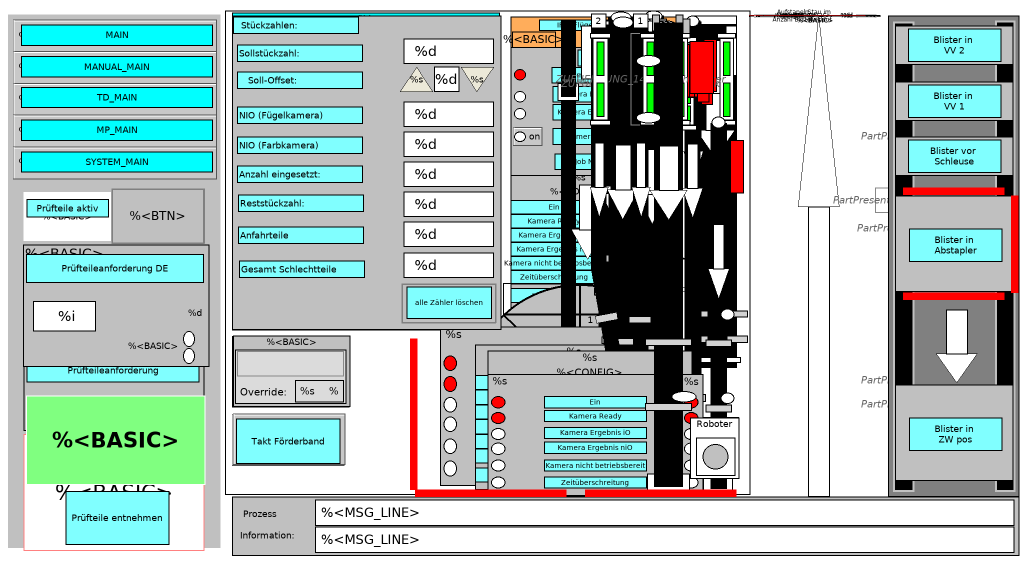
embedded screen at (220,111)-(745,597): ZUFUEHRUNG
rectangle at (227,597)-(1014,656): text "Prozess /  / Information:"
rectangle at (310,627)-(1009,653): text "%<MSG_LINE>"; shows ProcessMessage02; invisible if ProcessMessage02 = ''
rectangle at (310,600)-(1009,626): text "%<MSG_LINE>"; shows ProcessMessage01; invisible if ProcessMessage01=''
button at (228,514)-(340,565): text "%<BTN>"; shows 'TaktBand'; invisible if gTypeCode<>4991 AND gTypeCode <>312; taps ST03_Band.b_MoveRel; dynamic style Color.lightgrey, Color.grey
rectangle at (231,519)-(335,564): text "Takt Förderband"; invisible if TRUE
embedded screen at (744,116)-(875,597): WPC_Conveyor_Out
embedded screen at (898,492)-(923,517): PartPresentAndResult
embedded screen at (898,224)-(923,249): PartPresentAndResult
embedded screen at (3,115)-(215,648): M0000_Main
embedded screen at (898,468)-(923,493): PartPresentAndResult
embedded screen at (894,316)-(919,341): PartPresentAndResult
embedded screen at (870,288)-(895,313): PartPresentAndResult
embedded screen at (883,116)-(1014,597): WPC_CONVEYOR_IN
embedded screen at (18,283)-(204,651): PRUEFTEILENTNAHME
embedded screen at (227,116)-(496,430): TEILEZAEHLER
rectangle at (21,496)-(200,585): text "%<BASIC>"; shows 'Dummyprüfung aktiv'; invisible if NOT MP.ST02.DummyPruefung_93pol AND NOT DummyTest_160pol
rectangle at (228,436)-(345,507): text "%<BASIC>"; shows 'Föderband'; invisible if MP.ST03.SGM_3621
embedded screen at (230,450)-(341,504): ZLIB_OVERRIDE; invisible if MP.ST03.SGM_3621
rectangle at (685,518)-(734,579): text "Roboter"; opens MANUAL_ST03_0
embedded screen at (691,538)-(730,576): PARTRESULT; opens MANUAL_ST03_0
embedded screen at (410,590)-(561,597): DOOR_LOCK; tooltip ST00_220_S1_S31
embedded screen at (580,590)-(731,597): DOOR_LOCK; tooltip ST00_231_S1
embedded screen at (405,439)-(412,590): DOOR_LOCK; tooltip ST00_220_S2
*)

(* Visualisation MASTER_MAIN
embedded screen at (8,684)-(97,761): ZLIB_VISUBUTTON_MODE_SELECT
embedded screen at (100,684)-(189,761): ZLIB_VISUBUTTON_MODE_SELECT
embedded screen at (192,684)-(281,761): ZLIB_VISUBUTTON_MODE_SELECT
embedded screen at (284,684)-(373,761): ZLIB_VISUBUTTON_MODE_SELECT
embedded screen at (376,684)-(465,761): ZLIB_VISUBUTTON_MODE_SELECT
embedded screen at (468,684)-(557,761): ZLIB_VISUBUTTON_MODE_SELECT
embedded screen at (560,684)-(649,761): ZLIB_VISUBUTTON_MODE_SELECT
embedded screen at (652,684)-(741,761): ZLIB_VISUBUTTON_MODE_SELECT
embedded screen at (835,684)-(924,761): ZLIB_VISUBUTTON_MODE_SELECT
embedded screen at (927,684)-(1016,761): ZLIB_VISUBUTTON_MODE_SELECT
embedded screen at (4,655)-(1021,680): zLib_ErrorLine; opens zLib_ErrorHandler; dynamic style .Visu.ErrorHandler.Error[0].No<=1
rectangle at (388,29)-(673,49): text "%s"; shows .TD.ArtNo
rectangle at (247,29)-(386,49): text "%<DATA>:"; shows 'ArtNo'
rectangle at (388,6)-(673,26): text "%s"; shows .TD.TypeName
rectangle at (247,6)-(386,26): text "%<DATA>:"; shows 'TypeName'
rectangle at (388,52)-(673,72): text "%s"; shows .TD.TypeDescription
rectangle at (247,52)-(386,72): text "%<DATA>:"; shows 'TypeDescription'
rectangle at (9,50)-(241,73): text "User: %s"; shows UserLoginHandler.CurrentUser.UserName
embedded screen at (8,4)-(121,49): ZLIB_VISUBUTTON_S18; opens ZLIB_LOGIN
embedded screen at (120,4)-(242,49): ZLIB_VISUBUTTON_S18
rectangle at (13,81)-(243,101): text "%s"; shows CurrentVisu
embedded screen at (8,75)-(764,106): ZLIB_ShowMessageButton
embedded screen at (743,684)-(832,761): ZLIB_VISUBUTTON_MODE_SELECT
rectangle at (13,710)-(94,741): text "Manual"; invisible if TRUE
rectangle at (105,710)-(186,741): text "Auto"; invisible if TRUE
rectangle at (196,710)-(277,741): text "STEP"; invisible if TRUE
rectangle at (289,710)-(370,741): text "Autostart"; invisible if TRUE
rectangle at (381,710)-(462,741): text "Autostop"; invisible if TRUE
rectangle at (472,710)-(553,741): text "RunEmpty"; invisible if TRUE
rectangle at (564,710)-(645,741): text "StepCycle"; invisible if TRUE
rectangle at (657,710)-(738,741): text "Special"; invisible if TRUE
rectangle at (748,710)-(829,741): text "SpecStep"; invisible if TRUE
rectangle at (840,710)-(921,741): text "HomeRun"; invisible if TRUE
rectangle at (932,710)-(1013,741): text "Reset"; invisible if TRUE
rectangle at (142,11)-(223,42): text "LogOut"; invisible if TRUE
rectangle at (23,12)-(104,43): text "LogIn"; invisible if TRUE
rectangle at (157,52)-(239,71): text "%s"; shows UserLoginHandler.s_AutoLoggedOut
rectangle at (1,81)-(254,100): text "%s"; shows .gVarStrSystemTime
embedded screen at (168,2)-(253,46): MIN_EXIT; invisible if TRUE
embedded screen at (765,4)-(891,88): SPRACHE_MENUE
rounded rectangle at (0,0)-(91,40): text "%"; alarm colour if .MP.ST00.Override < .TD.Override_Robi
rounded rectangle at (1,0)-(73,40): text "Override: / %d"; shows .MP.ST00.Override; editable 2..100
6 more shapes without text or variables
*)

(* Visualisation M0000_MAIN
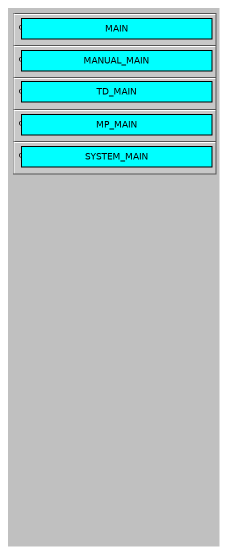
rectangle at (0,0)-(211,538): invisible if TRUE
embedded screen at (5,5)-(208,38): VISUBUTTON_TREE
embedded screen at (5,37)-(208,70): VISUBUTTON_TREE
embedded screen at (5,69)-(208,102): VISUBUTTON_TREE
embedded screen at (5,101)-(208,134): VISUBUTTON_TREE
embedded screen at (5,133)-(208,166): VISUBUTTON_TREE
rectangle at (13,10)-(204,31): text "MAIN"; invisible if TRUE
rectangle at (13,42)-(204,63): text "MANUAL_MAIN"; invisible if TRUE
rectangle at (13,73)-(204,94): text "TD_MAIN"; invisible if TRUE
rectangle at (13,106)-(204,127): text "MP_MAIN"; invisible if TRUE
rectangle at (13,138)-(204,159): text "SYSTEM_MAIN"; invisible if TRUE
*)

(* Visualisation M0000_MANUAL
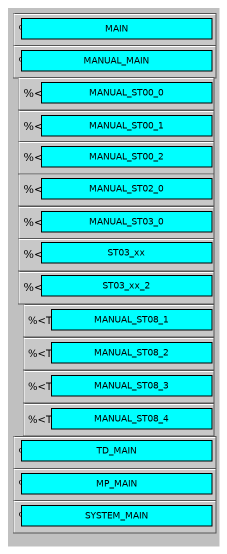
rectangle at (0,0)-(211,538): invisible if TRUE
embedded screen at (5,5)-(208,38): VISUBUTTON_TREE
embedded screen at (5,37)-(208,70): VISUBUTTON_TREE
embedded screen at (5,428)-(208,461): VISUBUTTON_TREE
embedded screen at (5,460)-(208,493): VISUBUTTON_TREE
embedded screen at (5,492)-(208,525): VISUBUTTON_TREE
rectangle at (13,10)-(204,31): text "MAIN"; invisible if TRUE
rectangle at (13,42)-(204,63): text "MANUAL_MAIN"; invisible if TRUE
rectangle at (13,432)-(204,453): text "TD_MAIN"; invisible if TRUE
rectangle at (13,465)-(204,486): text "MP_MAIN"; invisible if TRUE
rectangle at (13,497)-(204,518): text "SYSTEM_MAIN"; invisible if TRUE
embedded screen at (10,69)-(206,102): VISUBUTTON_TREE
rectangle at (33,74)-(204,95): text "MANUAL_ST00_0"; invisible if TRUE
embedded screen at (10,102)-(206,135): VISUBUTTON_TREE
rectangle at (33,107)-(204,128): text "MANUAL_ST00_1"; invisible if TRUE
embedded screen at (10,165)-(206,198): VISUBUTTON_TREE
rectangle at (33,170)-(204,191): text "MANUAL_ST02_0"; invisible if TRUE
embedded screen at (10,198)-(206,231): VISUBUTTON_TREE
rectangle at (33,203)-(204,224): text "MANUAL_ST03_0"; invisible if TRUE
embedded screen at (15,296)-(206,329): VISUBUTTON_TREE
rectangle at (43,301)-(204,322): text "MANUAL_ST08_1"; invisible if TRUE
embedded screen at (15,329)-(206,362): VISUBUTTON_TREE
rectangle at (43,334)-(204,355): text "MANUAL_ST08_2"; invisible if TRUE
embedded screen at (15,362)-(206,395): VISUBUTTON_TREE
rectangle at (43,367)-(204,388): text "MANUAL_ST08_3"; invisible if TRUE
embedded screen at (15,395)-(206,428): VISUBUTTON_TREE
rectangle at (43,400)-(204,421): text "MANUAL_ST08_4"; invisible if TRUE
embedded screen at (10,263)-(206,296): VISUBUTTON_TREE
embedded screen at (10,230)-(206,263): VISUBUTTON_TREE
rectangle at (33,267)-(204,288): text "ST03_xx_2"; invisible if TRUE
rectangle at (33,234)-(204,255): text "ST03_xx"; invisible if TRUE
embedded screen at (10,133)-(206,166): VISUBUTTON_TREE
rectangle at (33,138)-(204,159): text "MANUAL_ST00_2"; invisible if TRUE
*)

(* Visualisation M0002_MACHPARA
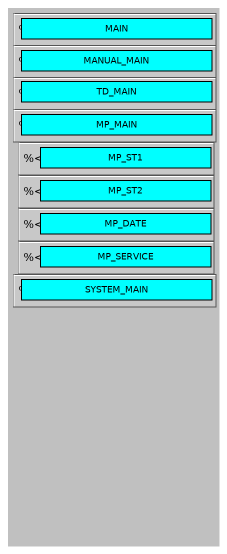
rectangle at (0,0)-(211,538): invisible if TRUE
embedded screen at (5,5)-(208,38): VISUBUTTON_TREE
embedded screen at (5,37)-(208,70): VISUBUTTON_TREE
embedded screen at (5,69)-(208,102): VISUBUTTON_TREE
embedded screen at (5,101)-(208,134): VISUBUTTON_TREE
embedded screen at (5,266)-(208,299): VISUBUTTON_TREE
rectangle at (13,10)-(204,31): text "MAIN"; invisible if TRUE
rectangle at (13,42)-(204,63): text "MANUAL_MAIN"; invisible if TRUE
rectangle at (13,73)-(204,94): text "TD_MAIN"; invisible if TRUE
rectangle at (13,106)-(204,127): text "MP_MAIN"; invisible if TRUE
rectangle at (13,271)-(204,292): text "SYSTEM_MAIN"; invisible if TRUE
embedded screen at (10,167)-(206,200): VISUBUTTON_TREE
rectangle at (32,172)-(203,193): text "MP_ST2"; invisible if TRUE
embedded screen at (10,200)-(206,233): VISUBUTTON_TREE
rectangle at (32,205)-(203,226): text "MP_DATE"; invisible if TRUE
embedded screen at (10,233)-(206,266): VISUBUTTON_TREE
rectangle at (32,238)-(203,259): text "MP_SERVICE"; invisible if TRUE
embedded screen at (10,134)-(206,167): VISUBUTTON_TREE
rectangle at (32,139)-(203,160): text "MP_ST1"; invisible if TRUE
*)

(* Visualisation M0003_SYSTEM
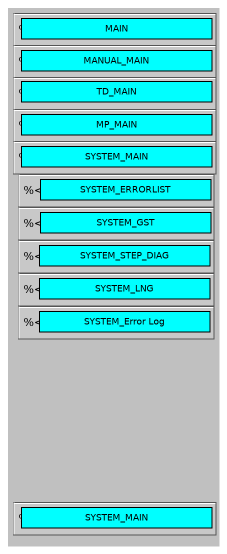
rectangle at (0,0)-(211,538): invisible if TRUE
embedded screen at (5,5)-(208,38): VISUBUTTON_TREE
embedded screen at (5,37)-(208,70): VISUBUTTON_TREE
embedded screen at (5,69)-(208,102): VISUBUTTON_TREE
embedded screen at (5,101)-(208,134): VISUBUTTON_TREE
embedded screen at (5,133)-(208,166): VISUBUTTON_TREE
rectangle at (13,10)-(204,31): text "MAIN"; invisible if TRUE
rectangle at (13,42)-(204,63): text "MANUAL_MAIN"; invisible if TRUE
rectangle at (13,73)-(204,94): text "TD_MAIN"; invisible if TRUE
rectangle at (13,106)-(204,127): text "MP_MAIN"; invisible if TRUE
rectangle at (13,138)-(204,159): text "SYSTEM_MAIN"; invisible if TRUE
embedded screen at (5,494)-(208,527): VISUBUTTON_TREE; invisible if TRUE; runs INTERN EXITPROGRAM
rectangle at (13,499)-(204,520): text "SYSTEM_MAIN"; invisible if TRUE
embedded screen at (10,166)-(206,199): VISUBUTTON_TREE
rectangle at (32,171)-(203,192): text "SYSTEM_ERRORLIST"; invisible if TRUE
embedded screen at (10,199)-(206,232): VISUBUTTON_TREE
rectangle at (32,204)-(203,225): text "SYSTEM_GST"; invisible if TRUE
embedded screen at (10,232)-(206,265): VISUBUTTON_TREE
rectangle at (31,237)-(202,258): text "SYSTEM_STEP_DIAG"; invisible if TRUE
embedded screen at (10,265)-(206,298): VISUBUTTON_TREE
rectangle at (31,270)-(202,291): text "SYSTEM_LNG"; invisible if TRUE
embedded screen at (10,298)-(206,331): VISUBUTTON_TREE
rectangle at (31,303)-(202,324): text "SYSTEM_Error Log"; invisible if TRUE
*)

(* Visualisation M0003_TD
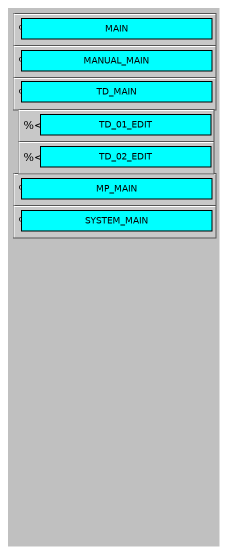
rectangle at (0,0)-(211,538): invisible if TRUE
embedded screen at (5,5)-(208,38): VISUBUTTON_TREE
embedded screen at (5,37)-(208,70): VISUBUTTON_TREE
embedded screen at (5,69)-(208,102): VISUBUTTON_TREE
embedded screen at (5,165)-(208,198): VISUBUTTON_TREE
embedded screen at (5,197)-(208,230): VISUBUTTON_TREE
rectangle at (13,10)-(204,31): text "MAIN"; invisible if TRUE
rectangle at (13,42)-(204,63): text "MANUAL_MAIN"; invisible if TRUE
rectangle at (13,73)-(204,94): text "TD_MAIN"; invisible if TRUE
rectangle at (13,170)-(204,191): text "MP_MAIN"; invisible if TRUE
rectangle at (13,202)-(204,223): text "SYSTEM_MAIN"; invisible if TRUE
embedded screen at (10,101)-(206,134): VISUBUTTON_TREE
rectangle at (32,106)-(203,127): text "TD_01_EDIT"; invisible if TRUE
embedded screen at (10,133)-(206,166): VISUBUTTON_TREE
rectangle at (32,138)-(203,159): text "TD_02_EDIT"; invisible if TRUE
*)

(* Visualisation MANUAL_MAIN
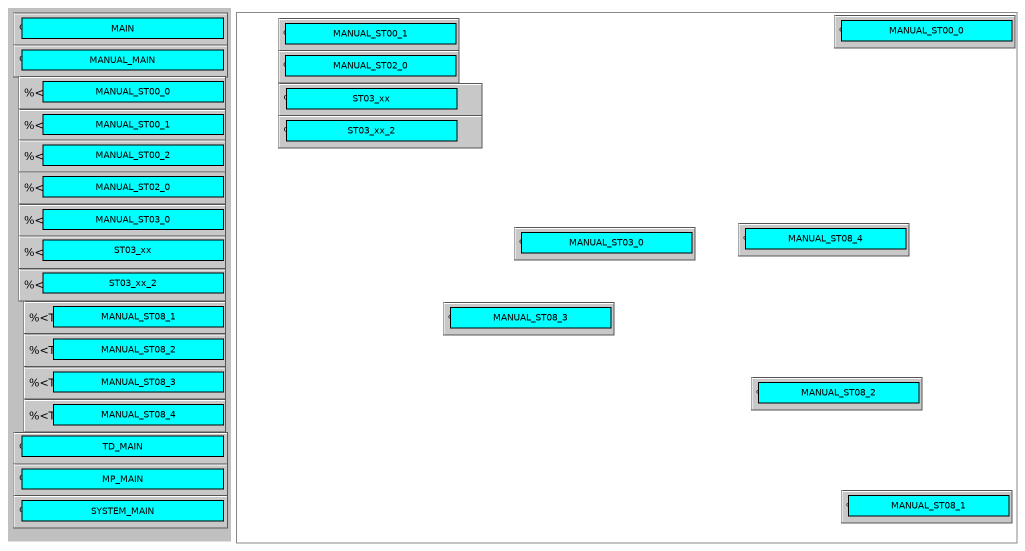
embedded screen at (3,115)-(226,648): M0000_Manual
embedded screen at (273,125)-(454,158): VISUBUTTON_TREE
rectangle at (280,130)-(451,151): text "MANUAL_ST00_1"; invisible if TRUE
embedded screen at (273,157)-(454,190): VISUBUTTON_TREE
rectangle at (280,162)-(451,183): text "MANUAL_ST02_0"; invisible if TRUE
embedded screen at (509,334)-(690,367): VISUBUTTON_TREE
rectangle at (516,339)-(687,360): text "MANUAL_ST03_0"; invisible if TRUE
embedded screen at (836,597)-(1007,630): VISUBUTTON_TREE
rectangle at (843,602)-(1004,623): text "MANUAL_ST08_1"; invisible if TRUE
embedded screen at (746,484)-(917,517): VISUBUTTON_TREE
rectangle at (753,489)-(914,510): text "MANUAL_ST08_2"; invisible if TRUE
embedded screen at (438,409)-(609,442): VISUBUTTON_TREE
rectangle at (445,414)-(606,435): text "MANUAL_ST08_3"; invisible if TRUE
embedded screen at (733,330)-(904,363): VISUBUTTON_TREE
rectangle at (740,335)-(901,356): text "MANUAL_ST08_4"; invisible if TRUE
embedded screen at (829,122)-(1010,155): VISUBUTTON_TREE
rectangle at (836,127)-(1007,148): text "MANUAL_ST00_0"; invisible if TRUE
embedded screen at (273,190)-(477,223): VISUBUTTON_TREE
rectangle at (281,195)-(452,216): text "ST03_xx"; invisible if TRUE
embedded screen at (273,222)-(477,255): VISUBUTTON_TREE
rectangle at (281,227)-(452,248): text "ST03_xx_2"; invisible if TRUE
1 more shapes without text or variables
*)

(* Visualisation MANUAL_ST00_0
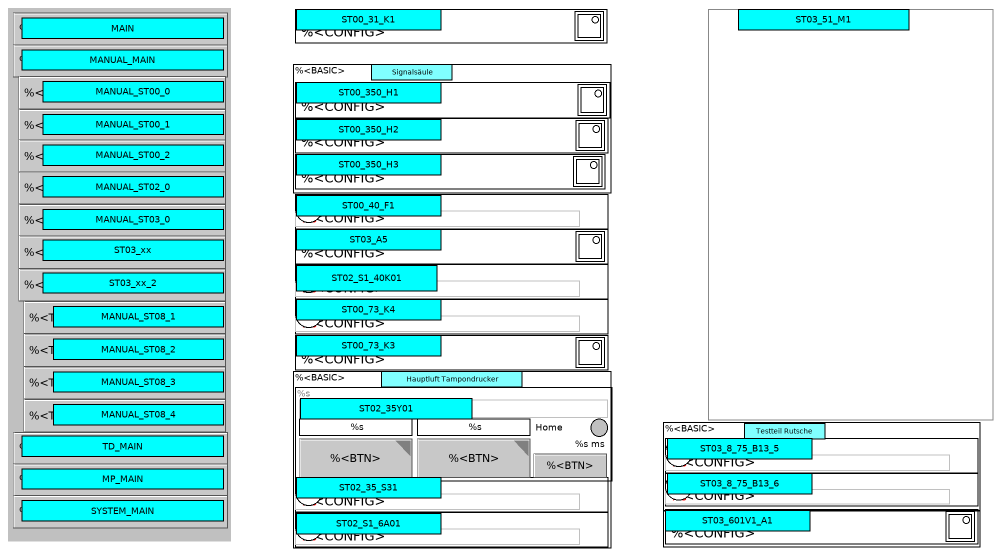
rectangle at (658,617)-(975,654): invisible if TD.TestpartBilister
embedded screen at (3,115)-(226,648): M0000_Manual
rectangle at (288,171)-(606,300): text "%<BASIC>"; shows 'Signalsäule'
embedded screen at (290,189)-(605,225): VDIGOUT_SMAL
embedded screen at (290,225)-(603,260): VDIGOUT_SMAL
embedded screen at (290,261)-(600,296): VDIGOUT_SMAL
embedded screen at (290,116)-(602,150): VDIGOUT_SMAL
embedded screen at (290,301)-(603,336): VDIGIN
other_LINEWIDTH at (703,116)-(988,527): invisible if MP.ST03.SGM_3621
embedded screen at (290,442)-(603,477): VDIGOUT_SMAL
rectangle at (288,478)-(606,655): text "%<BASIC>"; shows 'Tampondrucker'; invisible if gTypeCode<>4991 AND gTypeCode <>312
embedded screen at (290,584)-(603,619): VDIGIN; invisible if gTypeCode<>4991 AND gTypeCode <>312
embedded screen at (290,494)-(607,588): ZLIB_VALVE_1_SENSORS; invisible if gTypeCode<>4991 AND gTypeCode <>312
embedded screen at (290,619)-(603,654): VDIGIN; invisible if gTypeCode<>4991 AND gTypeCode <>312
rectangle at (658,529)-(975,618): text "%<BASIC>"; shows 'Testteil Rutsche'; invisible if TD.TestpartBilister
embedded screen at (660,545)-(973,580): VDIGIN; invisible if TD.TestpartBilister
embedded screen at (660,580)-(973,613): VDIGIN; invisible if TD.TestpartBilister
embedded screen at (290,336)-(603,371): VDIGOUT_SMAL; invisible if NOT MP.ST03.SGM_3621
rectangle at (739,530)-(820,546): text "Testteil Rutsche"; invisible if TRUE
rectangle at (366,171)-(447,187): text "Signalsäule"; invisible if TRUE
rectangle at (376,478)-(517,494): text "Hauptluft Tampondrucker"; invisible if TRUE
rectangle at (733,116)-(904,137): text "ST03_51_M1"; invisible if TRUE
embedded screen at (660,616)-(973,651): VDIGOUT_SMAL; invisible if NOT MP.ST03.BeltMotorCheckPartActive OR TD.TestpartBilister
rectangle at (295,505)-(467,526): text "ST02_35Y01"; invisible if TRUE
rectangle at (291,584)-(436,605): text "ST02_35_S31"; invisible if TRUE
rectangle at (291,620)-(436,641): text "ST02_S1_6A01"; invisible if TRUE
rectangle at (662,580)-(807,601): text "ST03_8_75_B13_6"; invisible if TRUE
rectangle at (662,545)-(807,566): text "ST03_8_75_B13_5"; invisible if TRUE
rectangle at (291,261)-(436,282): text "ST00_350_H3"; invisible if TRUE
rectangle at (291,442)-(436,463): text "ST00_73_K3"; invisible if TRUE
rectangle at (291,226)-(436,247): text "ST00_350_H2"; invisible if TRUE
rectangle at (291,189)-(436,210): text "ST00_350_H1"; invisible if TRUE
rectangle at (291,336)-(436,357): text "ST03_A5"; invisible if TRUE
rectangle at (660,617)-(805,638): text "ST03_601V1_A1"; invisible if TRUE
rectangle at (291,302)-(436,323): text "ST00_40_F1"; invisible if TRUE
rectangle at (291,116)-(436,137): text "ST00_31_K1"; invisible if TRUE
embedded screen at (290,406)-(603,441): VDIGIN
rectangle at (291,406)-(436,427): text "ST00_73_K4"; invisible if TRUE
embedded screen at (290,371)-(603,406): VDIGIN; invisible if gTypeCode<>4991 AND gTypeCode <>312
rectangle at (291,372)-(432,398): text "ST02_S1_40K01"; invisible if TRUE
*)

(* Visualisation MANUAL_ST00_1
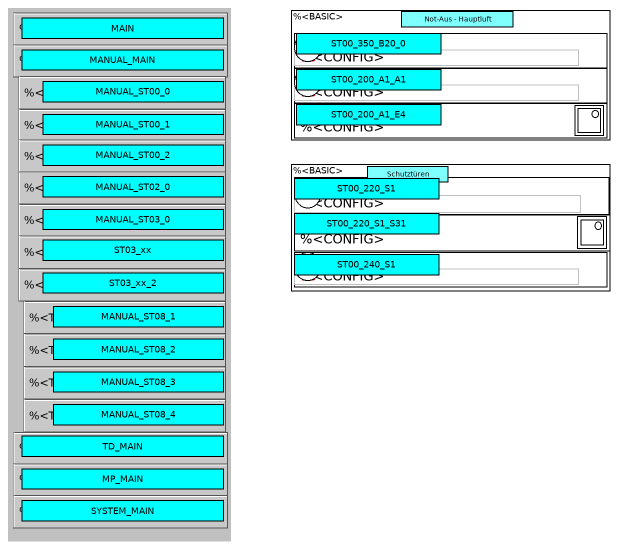
embedded screen at (3,115)-(226,648): M0000_Manual
rectangle at (286,271)-(605,398): text "%<BASIC>"; shows 'Schutztüren'
embedded screen at (289,321)-(605,358): VDIGOUT_SMAL
embedded screen at (289,284)-(604,322): VDIGIN
rectangle at (362,273)-(443,289): text "Schutztüren"; invisible if TRUE
rectangle at (289,320)-(434,341): text "ST00_220_S1_S31"; invisible if TRUE
rectangle at (289,285)-(434,306): text "ST00_220_S1"; invisible if TRUE
embedded screen at (289,359)-(602,394): VDIGIN
rectangle at (289,361)-(434,382): text "ST00_240_S1"; invisible if TRUE
rectangle at (286,117)-(605,247): text "%<BASIC>"; shows 'Not-Aus - Hauptluft'
embedded screen at (289,140)-(602,175): VDIGIN
embedded screen at (289,175)-(602,210): VDIGIN
embedded screen at (289,210)-(602,245): VDIGOUT_SMAL
rectangle at (396,118)-(508,134): text "Not-Aus - Hauptluft"; invisible if TRUE
rectangle at (291,140)-(436,161): text "ST00_350_B20_0"; invisible if TRUE
rectangle at (291,176)-(436,197): text "ST00_200_A1_A1"; invisible if TRUE
rectangle at (291,211)-(436,232): text "ST00_200_A1_E4"; invisible if TRUE
*)

